   1:  PR[GP1:91,1] = PR[GP1:90,1] + -10.638;
   1:  PR[GP1:91,2] = PR[GP1:90,2] + 34.723;
   1:L PR[91] 10mm/sec CNT100;
   1:  PR[GP1:91,1] = PR[GP1:90,1] + -15.376;
   1:  PR[GP1:91,2] = PR[GP1:90,2] + 36.085;
   1:L PR[91] 10mm/sec CNT100;
   1:  PR[GP1:91,1] = PR[GP1:90,1] + -20.922;
   1:  PR[GP1:91,2] = PR[GP1:90,2] + 37.394;
   1:L PR[91] 10mm/sec CNT100;
   1:  PR[GP1:91,1] = PR[GP1:90,1] + -26.137;
   1:  PR[GP1:91,2] = PR[GP1:90,2] + 37.739;
   1:L PR[91] 10mm/sec CNT100;
   1:  PR[GP1:91,1] = PR[GP1:90,1] + -31.979;
   1:  PR[GP1:91,2] = PR[GP1:90,2] + 36.930;
   1:L PR[91] 10mm/sec CNT100;
   1:  PR[GP1:91,1] = PR[GP1:90,1] + -36.500;
   1:  PR[GP1:91,2] = PR[GP1:90,2] + 36.505;
   1:L PR[91] 10mm/sec CNT100;
   1:  PR[GP1:91,1] = PR[GP1:90,1] + -42.224;
   1:  PR[GP1:91,2] = PR[GP1:90,2] + 34.409;
   1:L PR[91] 10mm/sec CNT100;
   1:  PR[GP1:91,1] = PR[GP1:90,1] + -45.685;
   1:  PR[GP1:91,2] = PR[GP1:90,2] + 32.896;
   1:L PR[91] 10mm/sec CNT100;
   1:  PR[GP1:91,1] = PR[GP1:90,1] + -50.990;
   1:  PR[GP1:91,2] = PR[GP1:90,2] + 29.551;
   1:L PR[91] 10mm/sec CNT100;
   1:  PR[GP1:91,1] = PR[GP1:90,1] + -55.793;
   1:  PR[GP1:91,2] = PR[GP1:90,2] + 24.861;
   1:L PR[91] 10mm/sec CNT100;
   1:  PR[GP1:91,1] = PR[GP1:90,1] + -57.811;
   1:  PR[GP1:91,2] = PR[GP1:90,2] + 23.034;
   1:L PR[91] 10mm/sec CNT100;
   1:  PR[GP1:91,1] = PR[GP1:90,1] + -61.510;
   1:  PR[GP1:91,2] = PR[GP1:90,2] + 17.261;
   1:L PR[91] 10mm/sec CNT100;
   1:  PR[GP1:91,1] = PR[GP1:90,1] + -62.600;
   1:  PR[GP1:91,2] = PR[GP1:90,2] + 15.293;
   1:L PR[91] 10mm/sec CNT100;
   1:  PR[GP1:91,1] = PR[GP1:90,1] + -64.933;
   1:  PR[GP1:91,2] = PR[GP1:90,2] + 8.866;
   1:L PR[91] 10mm/sec CNT100;
   1:  PR[GP1:91,1] = PR[GP1:90,1] + -65.686;
   1:  PR[GP1:91,2] = PR[GP1:90,2] + 2.142;
   1:L PR[91] 10mm/sec CNT100;
   1:  PR[GP1:91,1] = PR[GP1:90,1] + -66.007;
   1:  PR[GP1:91,2] = PR[GP1:90,2] + 0.261;
   1:L PR[91] 10mm/sec CNT100;
   1:  PR[GP1:91,1] = PR[GP1:90,1] + -65.270;
   1:  PR[GP1:91,2] = PR[GP1:90,2] + -6.357;
   1:L PR[91] 10mm/sec CNT100;
   1:  PR[GP1:91,1] = PR[GP1:90,1] + -64.940;
   1:  PR[GP1:91,2] = PR[GP1:90,2] + -8.287;
   1:L PR[91] 10mm/sec CNT100;
   1:  PR[GP1:91,1] = PR[GP1:90,1] + -62.601;
   1:  PR[GP1:91,2] = PR[GP1:90,2] + -14.731;
   1:L PR[91] 10mm/sec CNT100;
   1:  PR[GP1:91,1] = PR[GP1:90,1] + -61.517;
   1:  PR[GP1:91,2] = PR[GP1:90,2] + -16.695;
   1:L PR[91] 10mm/sec CNT100;
   1:  PR[GP1:91,1] = PR[GP1:90,1] + -57.812;
   1:  PR[GP1:91,2] = PR[GP1:90,2] + -22.477;
   1:L PR[91] 10mm/sec CNT100;
   1:  PR[GP1:91,1] = PR[GP1:90,1] + -53.300;
   1:  PR[GP1:91,2] = PR[GP1:90,2] + -26.904;
   1:L PR[91] 10mm/sec CNT100;
   1:  PR[GP1:91,1] = PR[GP1:90,1] + -51.017;
   1:  PR[GP1:91,2] = PR[GP1:90,2] + -28.975;
   1:L PR[91] 10mm/sec CNT100;
   1:  PR[GP1:91,1] = PR[GP1:90,1] + -45.704;
   1:  PR[GP1:91,2] = PR[GP1:90,2] + -32.325;
   1:L PR[91] 10mm/sec CNT100;
   1:  PR[GP1:91,1] = PR[GP1:90,1] + -42.257;
   1:  PR[GP1:91,2] = PR[GP1:90,2] + -33.842;
   1:L PR[91] 10mm/sec CNT100;
   1:  PR[GP1:91,1] = PR[GP1:90,1] + -36.523;
   1:  PR[GP1:91,2] = PR[GP1:90,2] + -35.942;
   1:L PR[91] 10mm/sec CNT100;
   1:  PR[GP1:91,1] = PR[GP1:90,1] + -31.071;
   1:  PR[GP1:91,2] = PR[GP1:90,2] + -36.718;
   1:L PR[91] 10mm/sec CNT100;
   1:  PR[GP1:91,1] = PR[GP1:90,1] + -26.206;
   1:  PR[GP1:91,2] = PR[GP1:90,2] + -37.185;
   1:L PR[91] 10mm/sec CNT100;
   1:  PR[GP1:91,1] = PR[GP1:90,1] + -20.979;
   1:  PR[GP1:91,2] = PR[GP1:90,2] + -36.840;
   1:L PR[91] 10mm/sec CNT100;
   1:  PR[GP1:91,1] = PR[GP1:90,1] + -15.524;
   1:  PR[GP1:91,2] = PR[GP1:90,2] + -35.592;
   1:L PR[91] 10mm/sec CNT100;
   1:  PR[GP1:91,1] = PR[GP1:90,1] + -10.757;
   1:  PR[GP1:91,2] = PR[GP1:90,2] + -34.223;
   1:L PR[91] 10mm/sec CNT100;
   1:  PR[GP1:91,1] = PR[GP1:90,1] + -5.971;
   1:  PR[GP1:91,2] = PR[GP1:90,2] + -31.419;
   1:L PR[91] 10mm/sec CNT100;
   1:  PR[GP1:91,1] = PR[GP1:90,1] + -3.818;
   1:  PR[GP1:91,2] = PR[GP1:90,2] + -30.247;
   1:L PR[91] 10mm/sec CNT100;
   1:  PR[GP1:91,1] = PR[GP1:90,1] + -0.263;
   1:  PR[GP1:91,2] = PR[GP1:90,2] + -27.179;
   1:L PR[91] 10mm/sec CNT100;
   1:  PR[GP1:91,1] = PR[GP1:90,1] + 3.052;
   1:  PR[GP1:91,2] = PR[GP1:90,2] + -30.324;
   1:  PR[GP1:91,3] = PR[GP1:90,3] + 60.695;
   1:L PR[91] 10mm/sec CNT100;
   1:  PR[GP1:91,1] = PR[GP1:90,1] + 5.026;
   1:  PR[GP1:91,2] = PR[GP1:90,2] + -31.395;
   1:L PR[91] 10mm/sec CNT100;
   1:  PR[GP1:91,1] = PR[GP1:90,1] + 9.972;
   1:  PR[GP1:91,2] = PR[GP1:90,2] + -34.290;
   1:L PR[91] 10mm/sec CNT100;
   1:  PR[GP1:91,1] = PR[GP1:90,1] + 14.624;
   1:  PR[GP1:91,2] = PR[GP1:90,2] + -35.626;
   1:L PR[91] 10mm/sec CNT100;
   1:  PR[GP1:91,1] = PR[GP1:90,1] + 20.278;
   1:  PR[GP1:91,2] = PR[GP1:90,2] + -36.920;
   1:L PR[91] 10mm/sec CNT100;
   1:  PR[GP1:91,1] = PR[GP1:90,1] + 25.353;
   1:  PR[GP1:91,2] = PR[GP1:90,2] + -37.257;
   1:L PR[91] 10mm/sec CNT100;
   1:  PR[GP1:91,1] = PR[GP1:90,1] + 31.035;
   1:  PR[GP1:91,2] = PR[GP1:90,2] + -36.473;
   1:L PR[91] 10mm/sec CNT100;
   1:  PR[GP1:91,1] = PR[GP1:90,1] + 35.762;
   1:  PR[GP1:91,2] = PR[GP1:90,2] + -36.013;
   1:L PR[91] 10mm/sec CNT100;
   1:  PR[GP1:91,1] = PR[GP1:90,1] + 41.363;
   1:  PR[GP1:91,2] = PR[GP1:90,2] + -33.969;
   1:L PR[91] 10mm/sec CNT100;
   1:  PR[GP1:91,1] = PR[GP1:90,1] + 45.011;
   1:  PR[GP1:91,2] = PR[GP1:90,2] + -32.365;
   1:L PR[91] 10mm/sec CNT100;
   1:  PR[GP1:91,1] = PR[GP1:90,1] + 50.172;
   1:  PR[GP1:91,2] = PR[GP1:90,2] + -29.127;
   1:L PR[91] 10mm/sec CNT100;
   1:  PR[GP1:91,1] = PR[GP1:90,1] + 54.865;
   1:  PR[GP1:91,2] = PR[GP1:90,2] + -24.552;
   1:L PR[91] 10mm/sec CNT100;
   1:  PR[GP1:91,1] = PR[GP1:90,1] + 57.047;
   1:  PR[GP1:91,2] = PR[GP1:90,2] + -22.568;
   1:L PR[91] 10mm/sec CNT100;
   1:  PR[GP1:91,1] = PR[GP1:90,1] + 60.710;
   1:  PR[GP1:91,2] = PR[GP1:90,2] + -16.886;
   1:L PR[91] 10mm/sec CNT100;
   1:  PR[GP1:91,1] = PR[GP1:90,1] + 61.903;
   1:  PR[GP1:91,2] = PR[GP1:90,2] + -14.729;
   1:L PR[91] 10mm/sec CNT100;
   1:  PR[GP1:91,1] = PR[GP1:90,1] + 64.181;
   1:  PR[GP1:91,2] = PR[GP1:90,2] + -8.537;
   1:L PR[91] 10mm/sec CNT100;
   1:  PR[GP1:91,1] = PR[GP1:90,1] + 64.946;
   1:  PR[GP1:91,2] = PR[GP1:90,2] + -1.801;
   1:L PR[91] 10mm/sec CNT100;
   1:  PR[GP1:91,1] = PR[GP1:90,1] + 65.304;
   1:  PR[GP1:91,2] = PR[GP1:90,2] + 0.296;
   1:L PR[91] 10mm/sec CNT100;
   1:  PR[GP1:91,1] = PR[GP1:90,1] + 64.554;
   1:  PR[GP1:91,2] = PR[GP1:90,2] + 6.927;
   1:L PR[91] 10mm/sec CNT100;
   1:  PR[GP1:91,1] = PR[GP1:90,1] + 64.185;
   1:  PR[GP1:91,2] = PR[GP1:90,2] + 9.083;
   1:L PR[91] 10mm/sec CNT100;
   1:  PR[GP1:91,1] = PR[GP1:90,1] + 61.901;
   1:  PR[GP1:91,2] = PR[GP1:90,2] + 15.292;
   1:L PR[91] 10mm/sec CNT100;
   1:  PR[GP1:91,1] = PR[GP1:90,1] + 60.703;
   1:  PR[GP1:91,2] = PR[GP1:90,2] + 17.452;
   1:L PR[91] 10mm/sec CNT100;
   1:  PR[GP1:91,1] = PR[GP1:90,1] + 57.033;
   1:  PR[GP1:91,2] = PR[GP1:90,2] + 23.145;
   1:L PR[91] 10mm/sec CNT100;
   1:  PR[GP1:91,1] = PR[GP1:90,1] + 52.617;
   1:  PR[GP1:91,2] = PR[GP1:90,2] + 27.469;
   1:L PR[91] 10mm/sec CNT100;
   1:  PR[GP1:91,1] = PR[GP1:90,1] + 50.162;
   1:  PR[GP1:91,2] = PR[GP1:90,2] + 29.691;
   1:L PR[91] 10mm/sec CNT100;
   1:  PR[GP1:91,1] = PR[GP1:90,1] + 44.991;
   1:  PR[GP1:91,2] = PR[GP1:90,2] + 32.936;
   1:L PR[91] 10mm/sec CNT100;
   1:  PR[GP1:91,1] = PR[GP1:90,1] + 41.328;
   1:  PR[GP1:91,2] = PR[GP1:90,2] + 34.536;
   1:L PR[91] 10mm/sec CNT100;
   1:  PR[GP1:91,1] = PR[GP1:90,1] + 35.711;
   1:  PR[GP1:91,2] = PR[GP1:90,2] + 36.586;
   1:L PR[91] 10mm/sec CNT100;
   1:  PR[GP1:91,1] = PR[GP1:90,1] + 30.393;
   1:  PR[GP1:91,2] = PR[GP1:90,2] + 37.340;
   1:L PR[91] 10mm/sec CNT100;
   1:  PR[GP1:91,1] = PR[GP1:90,1] + 25.308;
   1:  PR[GP1:91,2] = PR[GP1:90,2] + 37.812;
   1:L PR[91] 10mm/sec CNT100;
   1:  PR[GP1:91,1] = PR[GP1:90,1] + 20.219;
   1:  PR[GP1:91,2] = PR[GP1:90,2] + 37.474;
   1:L PR[91] 10mm/sec CNT100;
   1:  PR[GP1:91,1] = PR[GP1:90,1] + 14.472;
   1:  PR[GP1:91,2] = PR[GP1:90,2] + 36.117;
   1:L PR[91] 10mm/sec CNT100;
   1:  PR[GP1:91,1] = PR[GP1:90,1] + 9.851;
   1:  PR[GP1:91,2] = PR[GP1:90,2] + 34.788;
   1:L PR[91] 10mm/sec CNT100;
   1:  PR[GP1:91,1] = PR[GP1:90,1] + 5.551;
   1:  PR[GP1:91,2] = PR[GP1:90,2] + 32.480;
   1:L PR[91] 10mm/sec CNT100;
   1:  PR[GP1:91,1] = PR[GP1:90,1] + -0.263;
   1:  PR[GP1:91,2] = PR[GP1:90,2] + 27.751;
   1:L PR[91] 10mm/sec CNT100;
   1:  PR[GP1:91,1] = PR[GP1:90,1] + -6.062;
   1:  PR[GP1:91,2] = PR[GP1:90,2] + 32.466;
   1:L PR[91] 10mm/sec CNT100;
   1:  PR[GP1:91,1] = PR[GP1:90,1] + -10.379;
   1:  PR[GP1:91,2] = PR[GP1:90,2] + 34.791;
   1:L PR[91] 10mm/sec CNT100;
   1:  PR[GP1:91,1] = PR[GP1:90,1] + -14.995;
   1:  PR[GP1:91,2] = PR[GP1:90,2] + 36.117;
   1:L PR[91] 10mm/sec CNT100;
   1:  PR[GP1:91,1] = PR[GP1:90,1] + -20.743;
   1:  PR[GP1:91,2] = PR[GP1:90,2] + 37.475;
   1:L PR[91] 10mm/sec CNT100;
   1:  PR[GP1:91,1] = PR[GP1:90,1] + -25.835;
   1:  PR[GP1:91,2] = PR[GP1:90,2] + 37.810;
   1:L PR[91] 10mm/sec CNT100;
   1:  PR[GP1:91,1] = PR[GP1:90,1] + -31.540;
   1:  PR[GP1:91,2] = PR[GP1:90,2] + 37.021;
   1:L PR[91] 10mm/sec CNT100;
   1:  PR[GP1:91,1] = PR[GP1:90,1] + -36.280;
   1:  PR[GP1:91,2] = PR[GP1:90,2] + 36.575;
   1:L PR[91] 10mm/sec CNT100;
   1:  PR[GP1:91,1] = PR[GP1:90,1] + -41.877;
   1:  PR[GP1:91,2] = PR[GP1:90,2] + 34.525;
   1:L PR[91] 10mm/sec CNT100;
   1:  PR[GP1:91,1] = PR[GP1:90,1] + -45.538;
   1:  PR[GP1:91,2] = PR[GP1:90,2] + 32.925;
   1:L PR[91] 10mm/sec CNT100;
   1:  PR[GP1:91,1] = PR[GP1:90,1] + -50.732;
   1:  PR[GP1:91,2] = PR[GP1:90,2] + 29.650;
   1:L PR[91] 10mm/sec CNT100;
   1:  PR[GP1:91,1] = PR[GP1:90,1] + -55.436;
   1:  PR[GP1:91,2] = PR[GP1:90,2] + 25.058;
   1:L PR[91] 10mm/sec CNT100;
   1:  PR[GP1:91,1] = PR[GP1:90,1] + -57.623;
   1:  PR[GP1:91,2] = PR[GP1:90,2] + 23.078;
   1:L PR[91] 10mm/sec CNT100;
   1:  PR[GP1:91,1] = PR[GP1:90,1] + -61.248;
   1:  PR[GP1:91,2] = PR[GP1:90,2] + 17.420;
   1:L PR[91] 10mm/sec CNT100;
   1:  PR[GP1:91,1] = PR[GP1:90,1] + -62.445;
   1:  PR[GP1:91,2] = PR[GP1:90,2] + 15.257;
   1:L PR[91] 10mm/sec CNT100;
   1:  PR[GP1:91,1] = PR[GP1:90,1] + -64.732;
   1:  PR[GP1:91,2] = PR[GP1:90,2] + 8.956;
   1:L PR[91] 10mm/sec CNT100;
   1:  PR[GP1:91,1] = PR[GP1:90,1] + -65.471;
   1:  PR[GP1:91,2] = PR[GP1:90,2] + 2.362;
   1:L PR[91] 10mm/sec CNT100;
   1:  PR[GP1:91,1] = PR[GP1:90,1] + -65.830;
   1:  PR[GP1:91,2] = PR[GP1:90,2] + 0.261;
   1:L PR[91] 10mm/sec CNT100;
   1:  PR[GP1:91,1] = PR[GP1:90,1] + -65.107;
   1:  PR[GP1:91,2] = PR[GP1:90,2] + -6.229;
   1:L PR[91] 10mm/sec CNT100;
   1:  PR[GP1:91,1] = PR[GP1:90,1] + -64.740;
   1:  PR[GP1:91,2] = PR[GP1:90,2] + -8.377;
   1:L PR[91] 10mm/sec CNT100;
   1:  PR[GP1:91,1] = PR[GP1:90,1] + -62.447;
   1:  PR[GP1:91,2] = PR[GP1:90,2] + -14.694;
   1:L PR[91] 10mm/sec CNT100;
   1:  PR[GP1:91,1] = PR[GP1:90,1] + -61.255;
   1:  PR[GP1:91,2] = PR[GP1:90,2] + -16.853;
   1:L PR[91] 10mm/sec CNT100;
   1:  PR[GP1:91,1] = PR[GP1:90,1] + -57.624;
   1:  PR[GP1:91,2] = PR[GP1:90,2] + -22.520;
   1:L PR[91] 10mm/sec CNT100;
   1:  PR[GP1:91,1] = PR[GP1:90,1] + -53.202;
   1:  PR[GP1:91,2] = PR[GP1:90,2] + -26.858;
   1:L PR[91] 10mm/sec CNT100;
   1:  PR[GP1:91,1] = PR[GP1:90,1] + -50.760;
   1:  PR[GP1:91,2] = PR[GP1:90,2] + -29.074;
   1:L PR[91] 10mm/sec CNT100;
   1:  PR[GP1:91,1] = PR[GP1:90,1] + -45.558;
   1:  PR[GP1:91,2] = PR[GP1:90,2] + -32.353;
   1:L PR[91] 10mm/sec CNT100;
   1:  PR[GP1:91,1] = PR[GP1:90,1] + -41.912;
   1:  PR[GP1:91,2] = PR[GP1:90,2] + -33.958;
   1:L PR[91] 10mm/sec CNT100;
   1:  PR[GP1:91,1] = PR[GP1:90,1] + -36.305;
   1:  PR[GP1:91,2] = PR[GP1:90,2] + -36.012;
   1:L PR[91] 10mm/sec CNT100;
   1:  PR[GP1:91,1] = PR[GP1:90,1] + -30.973;
   1:  PR[GP1:91,2] = PR[GP1:90,2] + -36.771;
   1:L PR[91] 10mm/sec CNT100;
   1:  PR[GP1:91,1] = PR[GP1:90,1] + -25.905;
   1:  PR[GP1:91,2] = PR[GP1:90,2] + -37.257;
   1:L PR[91] 10mm/sec CNT100;
   1:  PR[GP1:91,1] = PR[GP1:90,1] + -20.802;
   1:  PR[GP1:91,2] = PR[GP1:90,2] + -36.920;
   1:L PR[91] 10mm/sec CNT100;
   1:  PR[GP1:91,1] = PR[GP1:90,1] + -15.149;
   1:  PR[GP1:91,2] = PR[GP1:90,2] + -35.627;
   1:L PR[91] 10mm/sec CNT100;
   1:  PR[GP1:91,1] = PR[GP1:90,1] + -10.503;
   1:  PR[GP1:91,2] = PR[GP1:90,2] + -34.292;
   1:L PR[91] 10mm/sec CNT100;
   1:  PR[GP1:91,1] = PR[GP1:90,1] + -5.560;
   1:  PR[GP1:91,2] = PR[GP1:90,2] + -31.397;
   1:L PR[91] 10mm/sec CNT100;
   1:  PR[GP1:91,1] = PR[GP1:90,1] + -3.575;
   1:  PR[GP1:91,2] = PR[GP1:90,2] + -30.316;
   1:L PR[91] 10mm/sec CNT100;
   1:  PR[GP1:91,1] = PR[GP1:90,1] + -0.263;
   1:  PR[GP1:91,2] = PR[GP1:90,2] + -27.459;
   1:L PR[91] 10mm/sec CNT100;
   1:  PR[GP1:91,1] = PR[GP1:90,1] + 2.808;
   1:  PR[GP1:91,2] = PR[GP1:90,2] + -30.392;
   1:  PR[GP1:91,3] = PR[GP1:90,3] + 61.305;
   1:L PR[91] 10mm/sec CNT100;
   1:  PR[GP1:91,1] = PR[GP1:90,1] + 4.615;
   1:  PR[GP1:91,2] = PR[GP1:90,2] + -31.374;
   1:L PR[91] 10mm/sec CNT100;
   1:  PR[GP1:91,1] = PR[GP1:90,1] + 9.717;
   1:  PR[GP1:91,2] = PR[GP1:90,2] + -34.360;
   1:L PR[91] 10mm/sec CNT100;
   1:  PR[GP1:91,1] = PR[GP1:90,1] + 14.249;
   1:  PR[GP1:91,2] = PR[GP1:90,2] + -35.661;
   1:L PR[91] 10mm/sec CNT100;
   1:  PR[GP1:91,1] = PR[GP1:90,1] + 20.101;
   1:  PR[GP1:91,2] = PR[GP1:90,2] + -37.000;
   1:L PR[91] 10mm/sec CNT100;
   1:  PR[GP1:91,1] = PR[GP1:90,1] + 25.053;
   1:  PR[GP1:91,2] = PR[GP1:90,2] + -37.329;
   1:L PR[91] 10mm/sec CNT100;
   1:  PR[GP1:91,1] = PR[GP1:90,1] + 30.599;
   1:  PR[GP1:91,2] = PR[GP1:90,2] + -36.563;
   1:L PR[91] 10mm/sec CNT100;
   1:  PR[GP1:91,1] = PR[GP1:90,1] + 35.544;
   1:  PR[GP1:91,2] = PR[GP1:90,2] + -36.083;
   1:L PR[91] 10mm/sec CNT100;
   1:  PR[GP1:91,1] = PR[GP1:90,1] + 41.019;
   1:  PR[GP1:91,2] = PR[GP1:90,2] + -34.085;
   1:L PR[91] 10mm/sec CNT100;
   1:  PR[GP1:91,1] = PR[GP1:90,1] + 44.866;
   1:  PR[GP1:91,2] = PR[GP1:90,2] + -32.393;
   1:L PR[91] 10mm/sec CNT100;
   1:  PR[GP1:91,1] = PR[GP1:90,1] + 49.916;
   1:  PR[GP1:91,2] = PR[GP1:90,2] + -29.224;
   1:L PR[91] 10mm/sec CNT100;
   1:  PR[GP1:91,1] = PR[GP1:90,1] + 54.510;
   1:  PR[GP1:91,2] = PR[GP1:90,2] + -24.747;
   1:L PR[91] 10mm/sec CNT100;
   1:  PR[GP1:91,1] = PR[GP1:90,1] + 56.860;
   1:  PR[GP1:91,2] = PR[GP1:90,2] + -22.610;
   1:L PR[91] 10mm/sec CNT100;
   1:  PR[GP1:91,1] = PR[GP1:90,1] + 60.448;
   1:  PR[GP1:91,2] = PR[GP1:90,2] + -17.043;
   1:L PR[91] 10mm/sec CNT100;
   1:  PR[GP1:91,1] = PR[GP1:90,1] + 61.749;
   1:  PR[GP1:91,2] = PR[GP1:90,2] + -14.692;
   1:L PR[91] 10mm/sec CNT100;
   1:  PR[GP1:91,1] = PR[GP1:90,1] + 63.981;
   1:  PR[GP1:91,2] = PR[GP1:90,2] + -8.624;
   1:L PR[91] 10mm/sec CNT100;
   1:  PR[GP1:91,1] = PR[GP1:90,1] + 64.731;
   1:  PR[GP1:91,2] = PR[GP1:90,2] + -2.021;
   1:L PR[91] 10mm/sec CNT100;
   1:  PR[GP1:91,1] = PR[GP1:90,1] + 65.127;
   1:  PR[GP1:91,2] = PR[GP1:90,2] + 0.296;
   1:L PR[91] 10mm/sec CNT100;
   1:  PR[GP1:91,1] = PR[GP1:90,1] + 64.392;
   1:  PR[GP1:91,2] = PR[GP1:90,2] + 6.797;
   1:L PR[91] 10mm/sec CNT100;
   1:  PR[GP1:91,1] = PR[GP1:90,1] + 63.985;
   1:  PR[GP1:91,2] = PR[GP1:90,2] + 9.171;
   1:L PR[91] 10mm/sec CNT100;
   1:  PR[GP1:91,1] = PR[GP1:90,1] + 61.747;
   1:  PR[GP1:91,2] = PR[GP1:90,2] + 15.256;
   1:L PR[91] 10mm/sec CNT100;
   1:  PR[GP1:91,1] = PR[GP1:90,1] + 60.441;
   1:  PR[GP1:91,2] = PR[GP1:90,2] + 17.611;
   1:L PR[91] 10mm/sec CNT100;
   1:  PR[GP1:91,1] = PR[GP1:90,1] + 56.845;
   1:  PR[GP1:91,2] = PR[GP1:90,2] + 23.188;
   1:L PR[91] 10mm/sec CNT100;
   1:  PR[GP1:91,1] = PR[GP1:90,1] + 52.520;
   1:  PR[GP1:91,2] = PR[GP1:90,2] + 27.423;
   1:L PR[91] 10mm/sec CNT100;
   1:  PR[GP1:91,1] = PR[GP1:90,1] + 49.906;
   1:  PR[GP1:91,2] = PR[GP1:90,2] + 29.789;
   1:L PR[91] 10mm/sec CNT100;
   1:  PR[GP1:91,1] = PR[GP1:90,1] + 44.844;
   1:  PR[GP1:91,2] = PR[GP1:90,2] + 32.965;
   1:L PR[91] 10mm/sec CNT100;
   1:  PR[GP1:91,1] = PR[GP1:90,1] + 40.982;
   1:  PR[GP1:91,2] = PR[GP1:90,2] + 34.652;
   1:L PR[91] 10mm/sec CNT100;
   1:  PR[GP1:91,1] = PR[GP1:90,1] + 35.492;
   1:  PR[GP1:91,2] = PR[GP1:90,2] + 36.656;
   1:L PR[91] 10mm/sec CNT100;
   1:  PR[GP1:91,1] = PR[GP1:90,1] + 30.294;
   1:  PR[GP1:91,2] = PR[GP1:90,2] + 37.393;
   1:L PR[91] 10mm/sec CNT100;
   1:  PR[GP1:91,1] = PR[GP1:90,1] + 25.006;
   1:  PR[GP1:91,2] = PR[GP1:90,2] + 37.884;
   1:L PR[91] 10mm/sec CNT100;
   1:  PR[GP1:91,1] = PR[GP1:90,1] + 20.040;
   1:  PR[GP1:91,2] = PR[GP1:90,2] + 37.554;
   1:L PR[91] 10mm/sec CNT100;
   1:  PR[GP1:91,1] = PR[GP1:90,1] + 14.092;
   1:  PR[GP1:91,2] = PR[GP1:90,2] + 36.149;
   1:L PR[91] 10mm/sec CNT100;
   1:  PR[GP1:91,1] = PR[GP1:90,1] + 9.593;
   1:  PR[GP1:91,2] = PR[GP1:90,2] + 34.856;
   1:L PR[91] 10mm/sec CNT100;
   1:  PR[GP1:91,1] = PR[GP1:90,1] + 5.378;
   1:  PR[GP1:91,2] = PR[GP1:90,2] + 32.594;
   1:L PR[91] 10mm/sec CNT100;
   1:  PR[GP1:91,1] = PR[GP1:90,1] + -0.263;
   1:  PR[GP1:91,2] = PR[GP1:90,2] + 28.006;
   1:L PR[91] 10mm/sec CNT100;
   1:  PR[GP1:91,1] = PR[GP1:90,1] + -5.889;
   1:  PR[GP1:91,2] = PR[GP1:90,2] + 32.580;
   1:L PR[91] 10mm/sec CNT100;
   1:  PR[GP1:91,1] = PR[GP1:90,1] + -10.121;
   1:  PR[GP1:91,2] = PR[GP1:90,2] + 34.858;
   1:L PR[91] 10mm/sec CNT100;
   1:  PR[GP1:91,1] = PR[GP1:90,1] + -14.614;
   1:  PR[GP1:91,2] = PR[GP1:90,2] + 36.150;
   1:L PR[91] 10mm/sec CNT100;
   1:  PR[GP1:91,1] = PR[GP1:90,1] + -20.564;
   1:  PR[GP1:91,2] = PR[GP1:90,2] + 37.555;
   1:L PR[91] 10mm/sec CNT100;
   1:  PR[GP1:91,1] = PR[GP1:90,1] + -25.532;
   1:  PR[GP1:91,2] = PR[GP1:90,2] + 37.882;
   1:L PR[91] 10mm/sec CNT100;
   1:  PR[GP1:91,1] = PR[GP1:90,1] + -31.101;
   1:  PR[GP1:91,2] = PR[GP1:90,2] + 37.112;
   1:L PR[91] 10mm/sec CNT100;
   1:  PR[GP1:91,1] = PR[GP1:90,1] + -36.060;
   1:  PR[GP1:91,2] = PR[GP1:90,2] + 36.645;
   1:L PR[91] 10mm/sec CNT100;
   1:  PR[GP1:91,1] = PR[GP1:90,1] + -41.531;
   1:  PR[GP1:91,2] = PR[GP1:90,2] + 34.642;
   1:L PR[91] 10mm/sec CNT100;
   1:  PR[GP1:91,1] = PR[GP1:90,1] + -45.391;
   1:  PR[GP1:91,2] = PR[GP1:90,2] + 32.954;
   1:L PR[91] 10mm/sec CNT100;
   1:  PR[GP1:91,1] = PR[GP1:90,1] + -50.474;
   1:  PR[GP1:91,2] = PR[GP1:90,2] + 29.749;
   1:L PR[91] 10mm/sec CNT100;
   1:  PR[GP1:91,1] = PR[GP1:90,1] + -55.078;
   1:  PR[GP1:91,2] = PR[GP1:90,2] + 25.255;
   1:L PR[91] 10mm/sec CNT100;
   1:  PR[GP1:91,1] = PR[GP1:90,1] + -57.434;
   1:  PR[GP1:91,2] = PR[GP1:90,2] + 23.121;
   1:L PR[91] 10mm/sec CNT100;
   1:  PR[GP1:91,1] = PR[GP1:90,1] + -60.985;
   1:  PR[GP1:91,2] = PR[GP1:90,2] + 17.579;
   1:L PR[91] 10mm/sec CNT100;
   1:  PR[GP1:91,1] = PR[GP1:90,1] + -62.290;
   1:  PR[GP1:91,2] = PR[GP1:90,2] + 15.221;
   1:L PR[91] 10mm/sec CNT100;
   1:  PR[GP1:91,1] = PR[GP1:90,1] + -64.532;
   1:  PR[GP1:91,2] = PR[GP1:90,2] + 9.045;
   1:L PR[91] 10mm/sec CNT100;
   1:  PR[GP1:91,1] = PR[GP1:90,1] + -65.256;
   1:  PR[GP1:91,2] = PR[GP1:90,2] + 2.582;
   1:L PR[91] 10mm/sec CNT100;
   1:  PR[GP1:91,1] = PR[GP1:90,1] + -65.653;
   1:  PR[GP1:91,2] = PR[GP1:90,2] + 0.261;
   1:L PR[91] 10mm/sec CNT100;
   1:  PR[GP1:91,1] = PR[GP1:90,1] + -64.944;
   1:  PR[GP1:91,2] = PR[GP1:90,2] + -6.101;
   1:L PR[91] 10mm/sec CNT100;
   1:  PR[GP1:91,1] = PR[GP1:90,1] + -64.540;
   1:  PR[GP1:91,2] = PR[GP1:90,2] + -8.466;
   1:L PR[91] 10mm/sec CNT100;
   1:  PR[GP1:91,1] = PR[GP1:90,1] + -62.292;
   1:  PR[GP1:91,2] = PR[GP1:90,2] + -14.658;
   1:L PR[91] 10mm/sec CNT100;
   1:  PR[GP1:91,1] = PR[GP1:90,1] + -60.993;
   1:  PR[GP1:91,2] = PR[GP1:90,2] + -17.012;
   1:L PR[91] 10mm/sec CNT100;
   1:  PR[GP1:91,1] = PR[GP1:90,1] + -57.436;
   1:  PR[GP1:91,2] = PR[GP1:90,2] + -22.563;
   1:L PR[91] 10mm/sec CNT100;
   1:  PR[GP1:91,1] = PR[GP1:90,1] + -53.104;
   1:  PR[GP1:91,2] = PR[GP1:90,2] + -26.813;
   1:L PR[91] 10mm/sec CNT100;
   1:  PR[GP1:91,1] = PR[GP1:90,1] + -50.503;
   1:  PR[GP1:91,2] = PR[GP1:90,2] + -29.172;
   1:L PR[91] 10mm/sec CNT100;
   1:  PR[GP1:91,1] = PR[GP1:90,1] + -45.413;
   1:  PR[GP1:91,2] = PR[GP1:90,2] + -32.382;
   1:L PR[91] 10mm/sec CNT100;
   1:  PR[GP1:91,1] = PR[GP1:90,1] + -41.568;
   1:  PR[GP1:91,2] = PR[GP1:90,2] + -34.074;
   1:L PR[91] 10mm/sec CNT100;
   1:  PR[GP1:91,1] = PR[GP1:90,1] + -36.087;
   1:  PR[GP1:91,2] = PR[GP1:90,2] + -36.082;
   1:L PR[91] 10mm/sec CNT100;
   1:  PR[GP1:91,1] = PR[GP1:90,1] + -30.875;
   1:  PR[GP1:91,2] = PR[GP1:90,2] + -36.823;
   1:L PR[91] 10mm/sec CNT100;
   1:  PR[GP1:91,1] = PR[GP1:90,1] + -25.605;
   1:  PR[GP1:91,2] = PR[GP1:90,2] + -37.329;
   1:L PR[91] 10mm/sec CNT100;
   1:  PR[GP1:91,1] = PR[GP1:90,1] + -20.626;
   1:  PR[GP1:91,2] = PR[GP1:90,2] + -37.000;
   1:L PR[91] 10mm/sec CNT100;
   1:  PR[GP1:91,1] = PR[GP1:90,1] + -14.773;
   1:  PR[GP1:91,2] = PR[GP1:90,2] + -35.661;
   1:L PR[91] 10mm/sec CNT100;
   1:  PR[GP1:91,1] = PR[GP1:90,1] + -10.248;
   1:  PR[GP1:91,2] = PR[GP1:90,2] + -34.362;
   1:L PR[91] 10mm/sec CNT100;
   1:  PR[GP1:91,1] = PR[GP1:90,1] + -5.149;
   1:  PR[GP1:91,2] = PR[GP1:90,2] + -31.375;
   1:L PR[91] 10mm/sec CNT100;
   1:  PR[GP1:91,1] = PR[GP1:90,1] + -3.331;
   1:  PR[GP1:91,2] = PR[GP1:90,2] + -30.385;
   1:L PR[91] 10mm/sec CNT100;
   1:  PR[GP1:91,1] = PR[GP1:90,1] + -0.264;
   1:  PR[GP1:91,2] = PR[GP1:90,2] + -27.738;
   1:L PR[91] 10mm/sec CNT100;
   1:  PR[GP1:91,1] = PR[GP1:90,1] + 2.563;
   1:  PR[GP1:91,2] = PR[GP1:90,2] + -30.461;
   1:  PR[GP1:91,3] = PR[GP1:90,3] + 61.915;
   1:L PR[91] 10mm/sec CNT100;
   1:  PR[GP1:91,1] = PR[GP1:90,1] + 4.205;
   1:  PR[GP1:91,2] = PR[GP1:90,2] + -31.352;
   1:L PR[91] 10mm/sec CNT100;
   1:  PR[GP1:91,1] = PR[GP1:90,1] + 9.463;
   1:  PR[GP1:91,2] = PR[GP1:90,2] + -34.429;
   1:L PR[91] 10mm/sec CNT100;
   1:  PR[GP1:91,1] = PR[GP1:90,1] + 13.873;
   1:  PR[GP1:91,2] = PR[GP1:90,2] + -35.696;
   1:L PR[91] 10mm/sec CNT100;
   1:  PR[GP1:91,1] = PR[GP1:90,1] + 19.924;
   1:  PR[GP1:91,2] = PR[GP1:90,2] + -37.080;
   1:L PR[91] 10mm/sec CNT100;
   1:  PR[GP1:91,1] = PR[GP1:90,1] + 24.753;
   1:  PR[GP1:91,2] = PR[GP1:90,2] + -37.401;
   1:L PR[91] 10mm/sec CNT100;
   1:  PR[GP1:91,1] = PR[GP1:90,1] + 30.163;
   1:  PR[GP1:91,2] = PR[GP1:90,2] + -36.654;
   1:L PR[91] 10mm/sec CNT100;
   1:  PR[GP1:91,1] = PR[GP1:90,1] + 35.327;
   1:  PR[GP1:91,2] = PR[GP1:90,2] + -36.152;
   1:L PR[91] 10mm/sec CNT100;
   1:  PR[GP1:91,1] = PR[GP1:90,1] + 40.675;
   1:  PR[GP1:91,2] = PR[GP1:90,2] + -34.200;
   1:L PR[91] 10mm/sec CNT100;
   1:  PR[GP1:91,1] = PR[GP1:90,1] + 44.721;
   1:  PR[GP1:91,2] = PR[GP1:90,2] + -32.421;
   1:L PR[91] 10mm/sec CNT100;
   1:  PR[GP1:91,1] = PR[GP1:90,1] + 49.661;
   1:  PR[GP1:91,2] = PR[GP1:90,2] + -29.322;
   1:L PR[91] 10mm/sec CNT100;
   1:  PR[GP1:91,1] = PR[GP1:90,1] + 54.155;
   1:  PR[GP1:91,2] = PR[GP1:90,2] + -24.942;
   1:L PR[91] 10mm/sec CNT100;
   1:  PR[GP1:91,1] = PR[GP1:90,1] + 56.673;
   1:  PR[GP1:91,2] = PR[GP1:90,2] + -22.651;
   1:L PR[91] 10mm/sec CNT100;
   1:  PR[GP1:91,1] = PR[GP1:90,1] + 60.187;
   1:  PR[GP1:91,2] = PR[GP1:90,2] + -17.201;
   1:L PR[91] 10mm/sec CNT100;
   1:  PR[GP1:91,1] = PR[GP1:90,1] + 61.595;
   1:  PR[GP1:91,2] = PR[GP1:90,2] + -14.656;
   1:L PR[91] 10mm/sec CNT100;
   1:  PR[GP1:91,1] = PR[GP1:90,1] + 63.781;
   1:  PR[GP1:91,2] = PR[GP1:90,2] + -8.710;
   1:L PR[91] 10mm/sec CNT100;
   1:  PR[GP1:91,1] = PR[GP1:90,1] + 64.517;
   1:  PR[GP1:91,2] = PR[GP1:90,2] + -2.241;
   1:L PR[91] 10mm/sec CNT100;
   1:  PR[GP1:91,1] = PR[GP1:90,1] + 64.949;
   1:  PR[GP1:91,2] = PR[GP1:90,2] + 0.296;
   1:L PR[91] 10mm/sec CNT100;
   1:  PR[GP1:91,1] = PR[GP1:90,1] + 64.229;
   1:  PR[GP1:91,2] = PR[GP1:90,2] + 6.666;
   1:L PR[91] 10mm/sec CNT100;
   1:  PR[GP1:91,1] = PR[GP1:90,1] + 63.785;
   1:  PR[GP1:91,2] = PR[GP1:90,2] + 9.258;
   1:L PR[91] 10mm/sec CNT100;
   1:  PR[GP1:91,1] = PR[GP1:90,1] + 61.593;
   1:  PR[GP1:91,2] = PR[GP1:90,2] + 15.219;
   1:L PR[91] 10mm/sec CNT100;
   1:  PR[GP1:91,1] = PR[GP1:90,1] + 60.179;
   1:  PR[GP1:91,2] = PR[GP1:90,2] + 17.769;
   1:L PR[91] 10mm/sec CNT100;
   1:  PR[GP1:91,1] = PR[GP1:90,1] + 56.658;
   1:  PR[GP1:91,2] = PR[GP1:90,2] + 23.230;
   1:L PR[91] 10mm/sec CNT100;
   1:  PR[GP1:91,1] = PR[GP1:90,1] + 52.422;
   1:  PR[GP1:91,2] = PR[GP1:90,2] + 27.377;
   1:L PR[91] 10mm/sec CNT100;
   1:  PR[GP1:91,1] = PR[GP1:90,1] + 49.649;
   1:  PR[GP1:91,2] = PR[GP1:90,2] + 29.888;
   1:L PR[91] 10mm/sec CNT100;
   1:  PR[GP1:91,1] = PR[GP1:90,1] + 44.698;
   1:  PR[GP1:91,2] = PR[GP1:90,2] + 32.994;
   1:L PR[91] 10mm/sec CNT100;
   1:  PR[GP1:91,1] = PR[GP1:90,1] + 40.636;
   1:  PR[GP1:91,2] = PR[GP1:90,2] + 34.769;
   1:L PR[91] 10mm/sec CNT100;
   1:  PR[GP1:91,1] = PR[GP1:90,1] + 35.272;
   1:  PR[GP1:91,2] = PR[GP1:90,2] + 36.726;
   1:L PR[91] 10mm/sec CNT100;
   1:  PR[GP1:91,1] = PR[GP1:90,1] + 30.195;
   1:  PR[GP1:91,2] = PR[GP1:90,2] + 37.446;
   1:L PR[91] 10mm/sec CNT100;
   1:  PR[GP1:91,1] = PR[GP1:90,1] + 24.704;
   1:  PR[GP1:91,2] = PR[GP1:90,2] + 37.956;
   1:L PR[91] 10mm/sec CNT100;
   1:  PR[GP1:91,1] = PR[GP1:90,1] + 19.861;
   1:  PR[GP1:91,2] = PR[GP1:90,2] + 37.634;
   1:L PR[91] 10mm/sec CNT100;
   1:  PR[GP1:91,1] = PR[GP1:90,1] + 13.711;
   1:  PR[GP1:91,2] = PR[GP1:90,2] + 36.182;
   1:L PR[91] 10mm/sec CNT100;
   1:  PR[GP1:91,1] = PR[GP1:90,1] + 9.334;
   1:  PR[GP1:91,2] = PR[GP1:90,2] + 34.924;
   1:L PR[91] 10mm/sec CNT100;
   1:  PR[GP1:91,1] = PR[GP1:90,1] + 5.205;
   1:  PR[GP1:91,2] = PR[GP1:90,2] + 32.708;
   1:L PR[91] 10mm/sec CNT100;
   1:  PR[GP1:91,1] = PR[GP1:90,1] + -0.263;
   1:  PR[GP1:91,2] = PR[GP1:90,2] + 28.260;
   1:L PR[91] 10mm/sec CNT100;
   1:  PR[GP1:91,1] = PR[GP1:90,1] + -5.717;
   1:  PR[GP1:91,2] = PR[GP1:90,2] + 32.695;
   1:L PR[91] 10mm/sec CNT100;
   1:  PR[GP1:91,1] = PR[GP1:90,1] + -9.863;
   1:  PR[GP1:91,2] = PR[GP1:90,2] + 34.926;
   1:L PR[91] 10mm/sec CNT100;
   1:  PR[GP1:91,1] = PR[GP1:90,1] + -14.233;
   1:  PR[GP1:91,2] = PR[GP1:90,2] + 36.182;
   1:L PR[91] 10mm/sec CNT100;
   1:  PR[GP1:91,1] = PR[GP1:90,1] + -20.386;
   1:  PR[GP1:91,2] = PR[GP1:90,2] + 37.635;
   1:L PR[91] 10mm/sec CNT100;
   1:  PR[GP1:91,1] = PR[GP1:90,1] + -25.230;
   1:  PR[GP1:91,2] = PR[GP1:90,2] + 37.954;
   1:L PR[91] 10mm/sec CNT100;
   1:  PR[GP1:91,1] = PR[GP1:90,1] + -30.661;
   1:  PR[GP1:91,2] = PR[GP1:90,2] + 37.202;
   1:L PR[91] 10mm/sec CNT100;
   1:  PR[GP1:91,1] = PR[GP1:90,1] + -35.840;
   1:  PR[GP1:91,2] = PR[GP1:90,2] + 36.716;
   1:L PR[91] 10mm/sec CNT100;
   1:  PR[GP1:91,1] = PR[GP1:90,1] + -41.184;
   1:  PR[GP1:91,2] = PR[GP1:90,2] + 34.758;
   1:L PR[91] 10mm/sec CNT100;
   1:  PR[GP1:91,1] = PR[GP1:90,1] + -45.244;
   1:  PR[GP1:91,2] = PR[GP1:90,2] + 32.983;
   1:L PR[91] 10mm/sec CNT100;
   1:  PR[GP1:91,1] = PR[GP1:90,1] + -50.216;
   1:  PR[GP1:91,2] = PR[GP1:90,2] + 29.849;
   1:L PR[91] 10mm/sec CNT100;
   1:  PR[GP1:91,1] = PR[GP1:90,1] + -54.720;
   1:  PR[GP1:91,2] = PR[GP1:90,2] + 25.451;
   1:L PR[91] 10mm/sec CNT100;
   1:  PR[GP1:91,1] = PR[GP1:90,1] + -57.245;
   1:  PR[GP1:91,2] = PR[GP1:90,2] + 23.165;
   1:L PR[91] 10mm/sec CNT100;
   1:  PR[GP1:91,1] = PR[GP1:90,1] + -60.722;
   1:  PR[GP1:91,2] = PR[GP1:90,2] + 17.738;
   1:L PR[91] 10mm/sec CNT100;
   1:  PR[GP1:91,1] = PR[GP1:90,1] + -62.136;
   1:  PR[GP1:91,2] = PR[GP1:90,2] + 15.185;
   1:L PR[91] 10mm/sec CNT100;
   1:  PR[GP1:91,1] = PR[GP1:90,1] + -64.332;
   1:  PR[GP1:91,2] = PR[GP1:90,2] + 9.135;
   1:L PR[91] 10mm/sec CNT100;
   1:  PR[GP1:91,1] = PR[GP1:90,1] + -65.041;
   1:  PR[GP1:91,2] = PR[GP1:90,2] + 2.802;
   1:L PR[91] 10mm/sec CNT100;
   1:  PR[GP1:91,1] = PR[GP1:90,1] + -65.476;
   1:  PR[GP1:91,2] = PR[GP1:90,2] + 0.261;
   1:L PR[91] 10mm/sec CNT100;
   1:  PR[GP1:91,1] = PR[GP1:90,1] + -64.781;
   1:  PR[GP1:91,2] = PR[GP1:90,2] + -5.973;
   1:L PR[91] 10mm/sec CNT100;
   1:  PR[GP1:91,1] = PR[GP1:90,1] + -64.340;
   1:  PR[GP1:91,2] = PR[GP1:90,2] + -8.555;
   1:L PR[91] 10mm/sec CNT100;
   1:  PR[GP1:91,1] = PR[GP1:90,1] + -62.138;
   1:  PR[GP1:91,2] = PR[GP1:90,2] + -14.622;
   1:L PR[91] 10mm/sec CNT100;
   1:  PR[GP1:91,1] = PR[GP1:90,1] + -60.730;
   1:  PR[GP1:91,2] = PR[GP1:90,2] + -17.170;
   1:L PR[91] 10mm/sec CNT100;
   1:  PR[GP1:91,1] = PR[GP1:90,1] + -57.248;
   1:  PR[GP1:91,2] = PR[GP1:90,2] + -22.606;
   1:L PR[91] 10mm/sec CNT100;
   1:  PR[GP1:91,1] = PR[GP1:90,1] + -53.006;
   1:  PR[GP1:91,2] = PR[GP1:90,2] + -26.767;
   1:L PR[91] 10mm/sec CNT100;
   1:  PR[GP1:91,1] = PR[GP1:90,1] + -50.247;
   1:  PR[GP1:91,2] = PR[GP1:90,2] + -29.271;
   1:L PR[91] 10mm/sec CNT100;
   1:  PR[GP1:91,1] = PR[GP1:90,1] + -45.267;
   1:  PR[GP1:91,2] = PR[GP1:90,2] + -32.410;
   1:L PR[91] 10mm/sec CNT100;
   1:  PR[GP1:91,1] = PR[GP1:90,1] + -41.223;
   1:  PR[GP1:91,2] = PR[GP1:90,2] + -34.190;
   1:L PR[91] 10mm/sec CNT100;
   1:  PR[GP1:91,1] = PR[GP1:90,1] + -35.869;
   1:  PR[GP1:91,2] = PR[GP1:90,2] + -36.152;
   1:L PR[91] 10mm/sec CNT100;
   1:  PR[GP1:91,1] = PR[GP1:90,1] + -30.777;
   1:  PR[GP1:91,2] = PR[GP1:90,2] + -36.876;
   1:L PR[91] 10mm/sec CNT100;
   1:  PR[GP1:91,1] = PR[GP1:90,1] + -25.305;
   1:  PR[GP1:91,2] = PR[GP1:90,2] + -37.401;
   1:L PR[91] 10mm/sec CNT100;
   1:  PR[GP1:91,1] = PR[GP1:90,1] + -20.449;
   1:  PR[GP1:91,2] = PR[GP1:90,2] + -37.081;
   1:L PR[91] 10mm/sec CNT100;
   1:  PR[GP1:91,1] = PR[GP1:90,1] + -14.398;
   1:  PR[GP1:91,2] = PR[GP1:90,2] + -35.696;
   1:L PR[91] 10mm/sec CNT100;
   1:  PR[GP1:91,1] = PR[GP1:90,1] + -9.993;
   1:  PR[GP1:91,2] = PR[GP1:90,2] + -34.431;
   1:L PR[91] 10mm/sec CNT100;
   1:  PR[GP1:91,1] = PR[GP1:90,1] + -4.739;
   1:  PR[GP1:91,2] = PR[GP1:90,2] + -31.353;
   1:L PR[91] 10mm/sec CNT100;
   1:  PR[GP1:91,1] = PR[GP1:90,1] + -3.088;
   1:  PR[GP1:91,2] = PR[GP1:90,2] + -30.454;
   1:L PR[91] 10mm/sec CNT100;
   1:  PR[GP1:91,1] = PR[GP1:90,1] + -0.264;
   1:  PR[GP1:91,2] = PR[GP1:90,2] + -28.017;
   1:L PR[91] 10mm/sec CNT100;
   1:  PR[GP1:91,1] = PR[GP1:90,1] + 2.319;
   1:  PR[GP1:91,2] = PR[GP1:90,2] + -30.529;
   1:  PR[GP1:91,3] = PR[GP1:90,3] + 62.525;
   1:L PR[91] 10mm/sec CNT100;
   1:  PR[GP1:91,1] = PR[GP1:90,1] + 3.794;
   1:  PR[GP1:91,2] = PR[GP1:90,2] + -31.330;
   1:L PR[91] 10mm/sec CNT100;
   1:  PR[GP1:91,1] = PR[GP1:90,1] + 9.208;
   1:  PR[GP1:91,2] = PR[GP1:90,2] + -34.498;
   1:L PR[91] 10mm/sec CNT100;
   1:  PR[GP1:91,1] = PR[GP1:90,1] + 13.498;
   1:  PR[GP1:91,2] = PR[GP1:90,2] + -35.731;
   1:L PR[91] 10mm/sec CNT100;
   1:  PR[GP1:91,1] = PR[GP1:90,1] + 19.748;
   1:  PR[GP1:91,2] = PR[GP1:90,2] + -37.161;
   1:L PR[91] 10mm/sec CNT100;
   1:  PR[GP1:91,1] = PR[GP1:90,1] + 24.453;
   1:  PR[GP1:91,2] = PR[GP1:90,2] + -37.473;
   1:L PR[91] 10mm/sec CNT100;
   1:  PR[GP1:91,1] = PR[GP1:90,1] + 29.727;
   1:  PR[GP1:91,2] = PR[GP1:90,2] + -36.745;
   1:L PR[91] 10mm/sec CNT100;
   1:  PR[GP1:91,1] = PR[GP1:90,1] + 35.109;
   1:  PR[GP1:91,2] = PR[GP1:90,2] + -36.222;
   1:L PR[91] 10mm/sec CNT100;
   1:  PR[GP1:91,1] = PR[GP1:90,1] + 40.331;
   1:  PR[GP1:91,2] = PR[GP1:90,2] + -34.316;
   1:L PR[91] 10mm/sec CNT100;
   1:  PR[GP1:91,1] = PR[GP1:90,1] + 44.576;
   1:  PR[GP1:91,2] = PR[GP1:90,2] + -32.449;
   1:L PR[91] 10mm/sec CNT100;
   1:  PR[GP1:91,1] = PR[GP1:90,1] + 49.405;
   1:  PR[GP1:91,2] = PR[GP1:90,2] + -29.419;
   1:L PR[91] 10mm/sec CNT100;
   1:  PR[GP1:91,1] = PR[GP1:90,1] + 53.800;
   1:  PR[GP1:91,2] = PR[GP1:90,2] + -25.136;
   1:L PR[91] 10mm/sec CNT100;
   1:  PR[GP1:91,1] = PR[GP1:90,1] + 56.486;
   1:  PR[GP1:91,2] = PR[GP1:90,2] + -22.693;
   1:L PR[91] 10mm/sec CNT100;
   1:  PR[GP1:91,1] = PR[GP1:90,1] + 59.925;
   1:  PR[GP1:91,2] = PR[GP1:90,2] + -17.358;
   1:L PR[91] 10mm/sec CNT100;
   1:  PR[GP1:91,1] = PR[GP1:90,1] + 61.441;
   1:  PR[GP1:91,2] = PR[GP1:90,2] + -14.619;
   1:L PR[91] 10mm/sec CNT100;
   1:  PR[GP1:91,1] = PR[GP1:90,1] + 63.582;
   1:  PR[GP1:91,2] = PR[GP1:90,2] + -8.797;
   1:L PR[91] 10mm/sec CNT100;
   1:  PR[GP1:91,1] = PR[GP1:90,1] + 64.302;
   1:  PR[GP1:91,2] = PR[GP1:90,2] + -2.461;
   1:L PR[91] 10mm/sec CNT100;
   1:  PR[GP1:91,1] = PR[GP1:90,1] + 64.772;
   1:  PR[GP1:91,2] = PR[GP1:90,2] + 0.296;
   1:L PR[91] 10mm/sec CNT100;
   1:  PR[GP1:91,1] = PR[GP1:90,1] + 64.067;
   1:  PR[GP1:91,2] = PR[GP1:90,2] + 6.535;
   1:L PR[91] 10mm/sec CNT100;
   1:  PR[GP1:91,1] = PR[GP1:90,1] + 63.586;
   1:  PR[GP1:91,2] = PR[GP1:90,2] + 9.345;
   1:L PR[91] 10mm/sec CNT100;
   1:  PR[GP1:91,1] = PR[GP1:90,1] + 61.439;
   1:  PR[GP1:91,2] = PR[GP1:90,2] + 15.183;
   1:L PR[91] 10mm/sec CNT100;
   1:  PR[GP1:91,1] = PR[GP1:90,1] + 59.916;
   1:  PR[GP1:91,2] = PR[GP1:90,2] + 17.927;
   1:L PR[91] 10mm/sec CNT100;
   1:  PR[GP1:91,1] = PR[GP1:90,1] + 56.470;
   1:  PR[GP1:91,2] = PR[GP1:90,2] + 23.272;
   1:L PR[91] 10mm/sec CNT100;
   1:  PR[GP1:91,1] = PR[GP1:90,1] + 52.325;
   1:  PR[GP1:91,2] = PR[GP1:90,2] + 27.331;
   1:L PR[91] 10mm/sec CNT100;
   1:  PR[GP1:91,1] = PR[GP1:90,1] + 49.392;
   1:  PR[GP1:91,2] = PR[GP1:90,2] + 29.986;
   1:L PR[91] 10mm/sec CNT100;
   1:  PR[GP1:91,1] = PR[GP1:90,1] + 44.552;
   1:  PR[GP1:91,2] = PR[GP1:90,2] + 33.023;
   1:L PR[91] 10mm/sec CNT100;
   1:  PR[GP1:91,1] = PR[GP1:90,1] + 40.290;
   1:  PR[GP1:91,2] = PR[GP1:90,2] + 34.885;
   1:L PR[91] 10mm/sec CNT100;
   1:  PR[GP1:91,1] = PR[GP1:90,1] + 35.053;
   1:  PR[GP1:91,2] = PR[GP1:90,2] + 36.796;
   1:L PR[91] 10mm/sec CNT100;
   1:  PR[GP1:91,1] = PR[GP1:90,1] + 30.096;
   1:  PR[GP1:91,2] = PR[GP1:90,2] + 37.499;
   1:L PR[91] 10mm/sec CNT100;
   1:  PR[GP1:91,1] = PR[GP1:90,1] + 24.402;
   1:  PR[GP1:91,2] = PR[GP1:90,2] + 38.028;
   1:L PR[91] 10mm/sec CNT100;
   1:  PR[GP1:91,1] = PR[GP1:90,1] + 19.683;
   1:  PR[GP1:91,2] = PR[GP1:90,2] + 37.714;
   1:L PR[91] 10mm/sec CNT100;
   1:  PR[GP1:91,1] = PR[GP1:90,1] + 13.330;
   1:  PR[GP1:91,2] = PR[GP1:90,2] + 36.214;
   1:L PR[91] 10mm/sec CNT100;
   1:  PR[GP1:91,1] = PR[GP1:90,1] + 9.076;
   1:  PR[GP1:91,2] = PR[GP1:90,2] + 34.991;
   1:L PR[91] 10mm/sec CNT100;
   1:  PR[GP1:91,1] = PR[GP1:90,1] + 5.032;
   1:  PR[GP1:91,2] = PR[GP1:90,2] + 32.822;
   1:L PR[91] 10mm/sec CNT100;
   1:  PR[GP1:91,1] = PR[GP1:90,1] + -0.263;
   1:  PR[GP1:91,2] = PR[GP1:90,2] + 28.515;
   1:L PR[91] 10mm/sec CNT100;
   1:  PR[GP1:91,1] = PR[GP1:90,1] + -5.545;
   1:  PR[GP1:91,2] = PR[GP1:90,2] + 32.810;
   1:L PR[91] 10mm/sec CNT100;
   1:  PR[GP1:91,1] = PR[GP1:90,1] + -8.723;
   1:  PR[GP1:91,2] = PR[GP1:90,2] + 34.531;
   1:L PR[91] 10mm/sec CNT100;
   1:  PR[GP1:91,1] = PR[GP1:90,1] + -9.602;
   1:  PR[GP1:91,2] = PR[GP1:90,2] + 34.992;
   1:L PR[91] 10mm/sec CNT100;
   1:  PR[GP1:91,1] = PR[GP1:90,1] + -13.852;
   1:  PR[GP1:91,2] = PR[GP1:90,2] + 36.215;
   1:L PR[91] 10mm/sec CNT100;
   1:  PR[GP1:91,1] = PR[GP1:90,1] + -20.207;
   1:  PR[GP1:91,2] = PR[GP1:90,2] + 37.715;
   1:L PR[91] 10mm/sec CNT100;
   1:  PR[GP1:91,1] = PR[GP1:90,1] + -24.927;
   1:  PR[GP1:91,2] = PR[GP1:90,2] + 38.026;
   1:L PR[91] 10mm/sec CNT100;
   1:  PR[GP1:91,1] = PR[GP1:90,1] + -30.222;
   1:  PR[GP1:91,2] = PR[GP1:90,2] + 37.293;
   1:L PR[91] 10mm/sec CNT100;
   1:  PR[GP1:91,1] = PR[GP1:90,1] + -35.620;
   1:  PR[GP1:91,2] = PR[GP1:90,2] + 36.786;
   1:L PR[91] 10mm/sec CNT100;
   1:  PR[GP1:91,1] = PR[GP1:90,1] + -40.838;
   1:  PR[GP1:91,2] = PR[GP1:90,2] + 34.875;
   1:L PR[91] 10mm/sec CNT100;
   1:  PR[GP1:91,1] = PR[GP1:90,1] + -45.098;
   1:  PR[GP1:91,2] = PR[GP1:90,2] + 33.012;
   1:L PR[91] 10mm/sec CNT100;
   1:  PR[GP1:91,1] = PR[GP1:90,1] + -49.958;
   1:  PR[GP1:91,2] = PR[GP1:90,2] + 29.948;
   1:L PR[91] 10mm/sec CNT100;
   1:  PR[GP1:91,1] = PR[GP1:90,1] + -54.363;
   1:  PR[GP1:91,2] = PR[GP1:90,2] + 25.648;
   1:L PR[91] 10mm/sec CNT100;
   1:  PR[GP1:91,1] = PR[GP1:90,1] + -57.057;
   1:  PR[GP1:91,2] = PR[GP1:90,2] + 23.209;
   1:L PR[91] 10mm/sec CNT100;
   1:  PR[GP1:91,1] = PR[GP1:90,1] + -60.460;
   1:  PR[GP1:91,2] = PR[GP1:90,2] + 17.898;
   1:L PR[91] 10mm/sec CNT100;
   1:  PR[GP1:91,1] = PR[GP1:90,1] + -61.981;
   1:  PR[GP1:91,2] = PR[GP1:90,2] + 15.149;
   1:L PR[91] 10mm/sec CNT100;
   1:  PR[GP1:91,1] = PR[GP1:90,1] + -64.131;
   1:  PR[GP1:91,2] = PR[GP1:90,2] + 9.225;
   1:L PR[91] 10mm/sec CNT100;
   1:  PR[GP1:91,1] = PR[GP1:90,1] + -64.826;
   1:  PR[GP1:91,2] = PR[GP1:90,2] + 3.022;
   1:L PR[91] 10mm/sec CNT100;
   1:  PR[GP1:91,1] = PR[GP1:90,1] + -65.299;
   1:  PR[GP1:91,2] = PR[GP1:90,2] + 0.261;
   1:L PR[91] 10mm/sec CNT100;
   1:  PR[GP1:91,1] = PR[GP1:90,1] + -64.618;
   1:  PR[GP1:91,2] = PR[GP1:90,2] + -5.845;
   1:L PR[91] 10mm/sec CNT100;
   1:  PR[GP1:91,1] = PR[GP1:90,1] + -64.139;
   1:  PR[GP1:91,2] = PR[GP1:90,2] + -8.644;
   1:L PR[91] 10mm/sec CNT100;
   1:  PR[GP1:91,1] = PR[GP1:90,1] + -61.983;
   1:  PR[GP1:91,2] = PR[GP1:90,2] + -14.585;
   1:L PR[91] 10mm/sec CNT100;
   1:  PR[GP1:91,1] = PR[GP1:90,1] + -60.468;
   1:  PR[GP1:91,2] = PR[GP1:90,2] + -17.328;
   1:L PR[91] 10mm/sec CNT100;
   1:  PR[GP1:91,1] = PR[GP1:90,1] + -57.060;
   1:  PR[GP1:91,2] = PR[GP1:90,2] + -22.649;
   1:L PR[91] 10mm/sec CNT100;
   1:  PR[GP1:91,1] = PR[GP1:90,1] + -52.909;
   1:  PR[GP1:91,2] = PR[GP1:90,2] + -26.721;
   1:L PR[91] 10mm/sec CNT100;
   1:  PR[GP1:91,1] = PR[GP1:90,1] + -49.990;
   1:  PR[GP1:91,2] = PR[GP1:90,2] + -29.369;
   1:L PR[91] 10mm/sec CNT100;
   1:  PR[GP1:91,1] = PR[GP1:90,1] + -45.122;
   1:  PR[GP1:91,2] = PR[GP1:90,2] + -32.439;
   1:L PR[91] 10mm/sec CNT100;
   1:  PR[GP1:91,1] = PR[GP1:90,1] + -40.878;
   1:  PR[GP1:91,2] = PR[GP1:90,2] + -34.306;
   1:L PR[91] 10mm/sec CNT100;
   1:  PR[GP1:91,1] = PR[GP1:90,1] + -35.651;
   1:  PR[GP1:91,2] = PR[GP1:90,2] + -36.221;
   1:L PR[91] 10mm/sec CNT100;
   1:  PR[GP1:91,1] = PR[GP1:90,1] + -30.679;
   1:  PR[GP1:91,2] = PR[GP1:90,2] + -36.929;
   1:L PR[91] 10mm/sec CNT100;
   1:  PR[GP1:91,1] = PR[GP1:90,1] + -25.005;
   1:  PR[GP1:91,2] = PR[GP1:90,2] + -37.473;
   1:L PR[91] 10mm/sec CNT100;
   1:  PR[GP1:91,1] = PR[GP1:90,1] + -20.272;
   1:  PR[GP1:91,2] = PR[GP1:90,2] + -37.161;
   1:L PR[91] 10mm/sec CNT100;
   1:  PR[GP1:91,1] = PR[GP1:90,1] + -14.023;
   1:  PR[GP1:91,2] = PR[GP1:90,2] + -35.731;
   1:L PR[91] 10mm/sec CNT100;
   1:  PR[GP1:91,1] = PR[GP1:90,1] + -9.738;
   1:  PR[GP1:91,2] = PR[GP1:90,2] + -34.501;
   1:L PR[91] 10mm/sec CNT100;
   1:  PR[GP1:91,1] = PR[GP1:90,1] + -4.328;
   1:  PR[GP1:91,2] = PR[GP1:90,2] + -31.331;
   1:L PR[91] 10mm/sec CNT100;
   1:  PR[GP1:91,1] = PR[GP1:90,1] + -2.844;
   1:  PR[GP1:91,2] = PR[GP1:90,2] + -30.523;
   1:L PR[91] 10mm/sec CNT100;
   1:  PR[GP1:91,1] = PR[GP1:90,1] + -0.264;
   1:  PR[GP1:91,2] = PR[GP1:90,2] + -28.297;
   1:L PR[91] 10mm/sec CNT100;
   1:  PR[GP1:91,1] = PR[GP1:90,1] + 2.074;
   1:  PR[GP1:91,2] = PR[GP1:90,2] + -30.597;
   1:  PR[GP1:91,3] = PR[GP1:90,3] + 63.135;
   1:L PR[91] 10mm/sec CNT100;
   1:  PR[GP1:91,1] = PR[GP1:90,1] + 3.384;
   1:  PR[GP1:91,2] = PR[GP1:90,2] + -31.308;
   1:L PR[91] 10mm/sec CNT100;
   1:  PR[GP1:91,1] = PR[GP1:90,1] + 8.953;
   1:  PR[GP1:91,2] = PR[GP1:90,2] + -34.568;
   1:L PR[91] 10mm/sec CNT100;
   1:  PR[GP1:91,1] = PR[GP1:90,1] + 13.123;
   1:  PR[GP1:91,2] = PR[GP1:90,2] + -35.765;
   1:L PR[91] 10mm/sec CNT100;
   1:  PR[GP1:91,1] = PR[GP1:90,1] + 19.571;
   1:  PR[GP1:91,2] = PR[GP1:90,2] + -37.241;
   1:L PR[91] 10mm/sec CNT100;
   1:  PR[GP1:91,1] = PR[GP1:90,1] + 24.153;
   1:  PR[GP1:91,2] = PR[GP1:90,2] + -37.545;
   1:L PR[91] 10mm/sec CNT100;
   1:  PR[GP1:91,1] = PR[GP1:90,1] + 29.291;
   1:  PR[GP1:91,2] = PR[GP1:90,2] + -36.836;
   1:L PR[91] 10mm/sec CNT100;
   1:  PR[GP1:91,1] = PR[GP1:90,1] + 34.892;
   1:  PR[GP1:91,2] = PR[GP1:90,2] + -36.292;
   1:L PR[91] 10mm/sec CNT100;
   1:  PR[GP1:91,1] = PR[GP1:90,1] + 39.987;
   1:  PR[GP1:91,2] = PR[GP1:90,2] + -34.432;
   1:L PR[91] 10mm/sec CNT100;
   1:  PR[GP1:91,1] = PR[GP1:90,1] + 44.430;
   1:  PR[GP1:91,2] = PR[GP1:90,2] + -32.478;
   1:L PR[91] 10mm/sec CNT100;
   1:  PR[GP1:91,1] = PR[GP1:90,1] + 49.150;
   1:  PR[GP1:91,2] = PR[GP1:90,2] + -29.517;
   1:L PR[91] 10mm/sec CNT100;
   1:  PR[GP1:91,1] = PR[GP1:90,1] + 53.445;
   1:  PR[GP1:91,2] = PR[GP1:90,2] + -25.331;
   1:L PR[91] 10mm/sec CNT100;
   1:  PR[GP1:91,1] = PR[GP1:90,1] + 56.299;
   1:  PR[GP1:91,2] = PR[GP1:90,2] + -22.734;
   1:L PR[91] 10mm/sec CNT100;
   1:  PR[GP1:91,1] = PR[GP1:90,1] + 59.663;
   1:  PR[GP1:91,2] = PR[GP1:90,2] + -17.516;
   1:L PR[91] 10mm/sec CNT100;
   1:  PR[GP1:91,1] = PR[GP1:90,1] + 61.287;
   1:  PR[GP1:91,2] = PR[GP1:90,2] + -14.582;
   1:L PR[91] 10mm/sec CNT100;
   1:  PR[GP1:91,1] = PR[GP1:90,1] + 63.382;
   1:  PR[GP1:91,2] = PR[GP1:90,2] + -8.884;
   1:L PR[91] 10mm/sec CNT100;
   1:  PR[GP1:91,1] = PR[GP1:90,1] + 64.087;
   1:  PR[GP1:91,2] = PR[GP1:90,2] + -2.680;
   1:L PR[91] 10mm/sec CNT100;
   1:  PR[GP1:91,1] = PR[GP1:90,1] + 64.595;
   1:  PR[GP1:91,2] = PR[GP1:90,2] + 0.296;
   1:L PR[91] 10mm/sec CNT100;
   1:  PR[GP1:91,1] = PR[GP1:90,1] + 63.904;
   1:  PR[GP1:91,2] = PR[GP1:90,2] + 6.405;
   1:L PR[91] 10mm/sec CNT100;
   1:  PR[GP1:91,1] = PR[GP1:90,1] + 63.386;
   1:  PR[GP1:91,2] = PR[GP1:90,2] + 9.432;
   1:L PR[91] 10mm/sec CNT100;
   1:  PR[GP1:91,1] = PR[GP1:90,1] + 61.284;
   1:  PR[GP1:91,2] = PR[GP1:90,2] + 15.146;
   1:L PR[91] 10mm/sec CNT100;
   1:  PR[GP1:91,1] = PR[GP1:90,1] + 59.654;
   1:  PR[GP1:91,2] = PR[GP1:90,2] + 18.086;
   1:L PR[91] 10mm/sec CNT100;
   1:  PR[GP1:91,1] = PR[GP1:90,1] + 56.283;
   1:  PR[GP1:91,2] = PR[GP1:90,2] + 23.314;
   1:L PR[91] 10mm/sec CNT100;
   1:  PR[GP1:91,1] = PR[GP1:90,1] + 52.228;
   1:  PR[GP1:91,2] = PR[GP1:90,2] + 27.286;
   1:L PR[91] 10mm/sec CNT100;
   1:  PR[GP1:91,1] = PR[GP1:90,1] + 49.135;
   1:  PR[GP1:91,2] = PR[GP1:90,2] + 30.084;
   1:L PR[91] 10mm/sec CNT100;
   1:  PR[GP1:91,1] = PR[GP1:90,1] + 44.405;
   1:  PR[GP1:91,2] = PR[GP1:90,2] + 33.052;
   1:L PR[91] 10mm/sec CNT100;
   1:  PR[GP1:91,1] = PR[GP1:90,1] + 39.944;
   1:  PR[GP1:91,2] = PR[GP1:90,2] + 35.001;
   1:L PR[91] 10mm/sec CNT100;
   1:  PR[GP1:91,1] = PR[GP1:90,1] + 34.834;
   1:  PR[GP1:91,2] = PR[GP1:90,2] + 36.866;
   1:L PR[91] 10mm/sec CNT100;
   1:  PR[GP1:91,1] = PR[GP1:90,1] + 29.996;
   1:  PR[GP1:91,2] = PR[GP1:90,2] + 37.552;
   1:L PR[91] 10mm/sec CNT100;
   1:  PR[GP1:91,1] = PR[GP1:90,1] + 24.099;
   1:  PR[GP1:91,2] = PR[GP1:90,2] + 38.100;
   1:L PR[91] 10mm/sec CNT100;
   1:  PR[GP1:91,1] = PR[GP1:90,1] + 19.504;
   1:  PR[GP1:91,2] = PR[GP1:90,2] + 37.795;
   1:L PR[91] 10mm/sec CNT100;
   1:  PR[GP1:91,1] = PR[GP1:90,1] + 12.949;
   1:  PR[GP1:91,2] = PR[GP1:90,2] + 36.247;
   1:L PR[91] 10mm/sec CNT100;
   1:  PR[GP1:91,1] = PR[GP1:90,1] + 8.816;
   1:  PR[GP1:91,2] = PR[GP1:90,2] + 35.058;
   1:L PR[91] 10mm/sec CNT100;
   1:  PR[GP1:91,1] = PR[GP1:90,1] + 7.908;
   1:  PR[GP1:91,2] = PR[GP1:90,2] + 34.582;
   1:L PR[91] 10mm/sec CNT100;
   1:  PR[GP1:91,1] = PR[GP1:90,1] + 4.860;
   1:  PR[GP1:91,2] = PR[GP1:90,2] + 32.936;
   1:L PR[91] 10mm/sec CNT100;
   1:  PR[GP1:91,1] = PR[GP1:90,1] + -0.263;
   1:  PR[GP1:91,2] = PR[GP1:90,2] + 28.770;
   1:L PR[91] 10mm/sec CNT100;
   1:  PR[GP1:91,1] = PR[GP1:90,1] + -5.373;
   1:  PR[GP1:91,2] = PR[GP1:90,2] + 32.924;
   1:L PR[91] 10mm/sec CNT100;
   1:  PR[GP1:91,1] = PR[GP1:90,1] + -8.438;
   1:  PR[GP1:91,2] = PR[GP1:90,2] + 34.584;
   1:L PR[91] 10mm/sec CNT100;
   1:  PR[GP1:91,1] = PR[GP1:90,1] + -9.344;
   1:  PR[GP1:91,2] = PR[GP1:90,2] + 35.060;
   1:L PR[91] 10mm/sec CNT100;
   1:  PR[GP1:91,1] = PR[GP1:90,1] + -13.472;
   1:  PR[GP1:91,2] = PR[GP1:90,2] + 36.247;
   1:L PR[91] 10mm/sec CNT100;
   1:  PR[GP1:91,1] = PR[GP1:90,1] + -20.028;
   1:  PR[GP1:91,2] = PR[GP1:90,2] + 37.795;
   1:L PR[91] 10mm/sec CNT100;
   1:  PR[GP1:91,1] = PR[GP1:90,1] + -24.624;
   1:  PR[GP1:91,2] = PR[GP1:90,2] + 38.098;
   1:L PR[91] 10mm/sec CNT100;
   1:  PR[GP1:91,1] = PR[GP1:90,1] + -29.783;
   1:  PR[GP1:91,2] = PR[GP1:90,2] + 37.384;
   1:L PR[91] 10mm/sec CNT100;
   1:  PR[GP1:91,1] = PR[GP1:90,1] + -35.400;
   1:  PR[GP1:91,2] = PR[GP1:90,2] + 36.856;
   1:L PR[91] 10mm/sec CNT100;
   1:  PR[GP1:91,1] = PR[GP1:90,1] + -40.491;
   1:  PR[GP1:91,2] = PR[GP1:90,2] + 34.992;
   1:L PR[91] 10mm/sec CNT100;
   1:  PR[GP1:91,1] = PR[GP1:90,1] + -44.951;
   1:  PR[GP1:91,2] = PR[GP1:90,2] + 33.042;
   1:L PR[91] 10mm/sec CNT100;
   1:  PR[GP1:91,1] = PR[GP1:90,1] + -49.700;
   1:  PR[GP1:91,2] = PR[GP1:90,2] + 30.047;
   1:L PR[91] 10mm/sec CNT100;
   1:  PR[GP1:91,1] = PR[GP1:90,1] + -54.005;
   1:  PR[GP1:91,2] = PR[GP1:90,2] + 25.844;
   1:L PR[91] 10mm/sec CNT100;
   1:  PR[GP1:91,1] = PR[GP1:90,1] + -56.868;
   1:  PR[GP1:91,2] = PR[GP1:90,2] + 23.252;
   1:L PR[91] 10mm/sec CNT100;
   1:  PR[GP1:91,1] = PR[GP1:90,1] + -60.197;
   1:  PR[GP1:91,2] = PR[GP1:90,2] + 18.057;
   1:L PR[91] 10mm/sec CNT100;
   1:  PR[GP1:91,1] = PR[GP1:90,1] + -61.826;
   1:  PR[GP1:91,2] = PR[GP1:90,2] + 15.113;
   1:L PR[91] 10mm/sec CNT100;
   1:  PR[GP1:91,1] = PR[GP1:90,1] + -63.931;
   1:  PR[GP1:91,2] = PR[GP1:90,2] + 9.315;
   1:L PR[91] 10mm/sec CNT100;
   1:  PR[GP1:91,1] = PR[GP1:90,1] + -64.611;
   1:  PR[GP1:91,2] = PR[GP1:90,2] + 3.242;
   1:L PR[91] 10mm/sec CNT100;
   1:  PR[GP1:91,1] = PR[GP1:90,1] + -65.121;
   1:  PR[GP1:91,2] = PR[GP1:90,2] + 0.261;
   1:L PR[91] 10mm/sec CNT100;
   1:  PR[GP1:91,1] = PR[GP1:90,1] + -64.455;
   1:  PR[GP1:91,2] = PR[GP1:90,2] + -5.717;
   1:L PR[91] 10mm/sec CNT100;
   1:  PR[GP1:91,1] = PR[GP1:90,1] + -63.939;
   1:  PR[GP1:91,2] = PR[GP1:90,2] + -8.734;
   1:L PR[91] 10mm/sec CNT100;
   1:  PR[GP1:91,1] = PR[GP1:90,1] + -61.829;
   1:  PR[GP1:91,2] = PR[GP1:90,2] + -14.549;
   1:L PR[91] 10mm/sec CNT100;
   1:  PR[GP1:91,1] = PR[GP1:90,1] + -60.206;
   1:  PR[GP1:91,2] = PR[GP1:90,2] + -17.487;
   1:L PR[91] 10mm/sec CNT100;
   1:  PR[GP1:91,1] = PR[GP1:90,1] + -56.872;
   1:  PR[GP1:91,2] = PR[GP1:90,2] + -22.692;
   1:L PR[91] 10mm/sec CNT100;
   1:  PR[GP1:91,1] = PR[GP1:90,1] + -52.811;
   1:  PR[GP1:91,2] = PR[GP1:90,2] + -26.676;
   1:L PR[91] 10mm/sec CNT100;
   1:  PR[GP1:91,1] = PR[GP1:90,1] + -49.733;
   1:  PR[GP1:91,2] = PR[GP1:90,2] + -29.468;
   1:L PR[91] 10mm/sec CNT100;
   1:  PR[GP1:91,1] = PR[GP1:90,1] + -44.976;
   1:  PR[GP1:91,2] = PR[GP1:90,2] + -32.467;
   1:L PR[91] 10mm/sec CNT100;
   1:  PR[GP1:91,1] = PR[GP1:90,1] + -40.534;
   1:  PR[GP1:91,2] = PR[GP1:90,2] + -34.422;
   1:L PR[91] 10mm/sec CNT100;
   1:  PR[GP1:91,1] = PR[GP1:90,1] + -35.432;
   1:  PR[GP1:91,2] = PR[GP1:90,2] + -36.291;
   1:L PR[91] 10mm/sec CNT100;
   1:  PR[GP1:91,1] = PR[GP1:90,1] + -30.581;
   1:  PR[GP1:91,2] = PR[GP1:90,2] + -36.981;
   1:L PR[91] 10mm/sec CNT100;
   1:  PR[GP1:91,1] = PR[GP1:90,1] + -24.704;
   1:  PR[GP1:91,2] = PR[GP1:90,2] + -37.545;
   1:L PR[91] 10mm/sec CNT100;
   1:  PR[GP1:91,1] = PR[GP1:90,1] + -20.095;
   1:  PR[GP1:91,2] = PR[GP1:90,2] + -37.241;
   1:L PR[91] 10mm/sec CNT100;
   1:  PR[GP1:91,1] = PR[GP1:90,1] + -13.647;
   1:  PR[GP1:91,2] = PR[GP1:90,2] + -35.766;
   1:L PR[91] 10mm/sec CNT100;
   1:  PR[GP1:91,1] = PR[GP1:90,1] + -9.484;
   1:  PR[GP1:91,2] = PR[GP1:90,2] + -34.570;
   1:L PR[91] 10mm/sec CNT100;
   1:  PR[GP1:91,1] = PR[GP1:90,1] + -3.918;
   1:  PR[GP1:91,2] = PR[GP1:90,2] + -31.309;
   1:L PR[91] 10mm/sec CNT100;
   1:  PR[GP1:91,1] = PR[GP1:90,1] + -2.601;
   1:  PR[GP1:91,2] = PR[GP1:90,2] + -30.592;
   1:L PR[91] 10mm/sec CNT100;
   1:  PR[GP1:91,1] = PR[GP1:90,1] + -0.264;
   1:  PR[GP1:91,2] = PR[GP1:90,2] + -28.576;
   1:L PR[91] 10mm/sec CNT100;
   1:  PR[GP1:91,1] = PR[GP1:90,1] + 1.830;
   1:  PR[GP1:91,2] = PR[GP1:90,2] + -30.666;
   1:  PR[GP1:91,3] = PR[GP1:90,3] + 63.745;
   1:L PR[91] 10mm/sec CNT100;
   1:  PR[GP1:91,1] = PR[GP1:90,1] + 2.973;
   1:  PR[GP1:91,2] = PR[GP1:90,2] + -31.286;
   1:L PR[91] 10mm/sec CNT100;
   1:  PR[GP1:91,1] = PR[GP1:90,1] + 8.699;
   1:  PR[GP1:91,2] = PR[GP1:90,2] + -34.637;
   1:L PR[91] 10mm/sec CNT100;
   1:  PR[GP1:91,1] = PR[GP1:90,1] + 12.747;
   1:  PR[GP1:91,2] = PR[GP1:90,2] + -35.800;
   1:L PR[91] 10mm/sec CNT100;
   1:  PR[GP1:91,1] = PR[GP1:90,1] + 19.394;
   1:  PR[GP1:91,2] = PR[GP1:90,2] + -37.321;
   1:L PR[91] 10mm/sec CNT100;
   1:  PR[GP1:91,1] = PR[GP1:90,1] + 23.853;
   1:  PR[GP1:91,2] = PR[GP1:90,2] + -37.617;
   1:L PR[91] 10mm/sec CNT100;
   1:  PR[GP1:91,1] = PR[GP1:90,1] + 28.855;
   1:  PR[GP1:91,2] = PR[GP1:90,2] + -36.927;
   1:L PR[91] 10mm/sec CNT100;
   1:  PR[GP1:91,1] = PR[GP1:90,1] + 34.674;
   1:  PR[GP1:91,2] = PR[GP1:90,2] + -36.361;
   1:L PR[91] 10mm/sec CNT100;
   1:  PR[GP1:91,1] = PR[GP1:90,1] + 39.642;
   1:  PR[GP1:91,2] = PR[GP1:90,2] + -34.548;
   1:L PR[91] 10mm/sec CNT100;
   1:  PR[GP1:91,1] = PR[GP1:90,1] + 44.285;
   1:  PR[GP1:91,2] = PR[GP1:90,2] + -32.506;
   1:L PR[91] 10mm/sec CNT100;
   1:  PR[GP1:91,1] = PR[GP1:90,1] + 48.894;
   1:  PR[GP1:91,2] = PR[GP1:90,2] + -29.614;
   1:L PR[91] 10mm/sec CNT100;
   1:  PR[GP1:91,1] = PR[GP1:90,1] + 53.090;
   1:  PR[GP1:91,2] = PR[GP1:90,2] + -25.525;
   1:L PR[91] 10mm/sec CNT100;
   1:  PR[GP1:91,1] = PR[GP1:90,1] + 56.112;
   1:  PR[GP1:91,2] = PR[GP1:90,2] + -22.776;
   1:L PR[91] 10mm/sec CNT100;
   1:  PR[GP1:91,1] = PR[GP1:90,1] + 59.402;
   1:  PR[GP1:91,2] = PR[GP1:90,2] + -17.674;
   1:L PR[91] 10mm/sec CNT100;
   1:  PR[GP1:91,1] = PR[GP1:90,1] + 61.132;
   1:  PR[GP1:91,2] = PR[GP1:90,2] + -14.545;
   1:L PR[91] 10mm/sec CNT100;
   1:  PR[GP1:91,1] = PR[GP1:90,1] + 63.183;
   1:  PR[GP1:91,2] = PR[GP1:90,2] + -8.971;
   1:L PR[91] 10mm/sec CNT100;
   1:  PR[GP1:91,1] = PR[GP1:90,1] + 63.873;
   1:  PR[GP1:91,2] = PR[GP1:90,2] + -2.900;
   1:L PR[91] 10mm/sec CNT100;
   1:  PR[GP1:91,1] = PR[GP1:90,1] + 64.418;
   1:  PR[GP1:91,2] = PR[GP1:90,2] + 0.296;
   1:L PR[91] 10mm/sec CNT100;
   1:  PR[GP1:91,1] = PR[GP1:90,1] + 63.742;
   1:  PR[GP1:91,2] = PR[GP1:90,2] + 6.274;
   1:L PR[91] 10mm/sec CNT100;
   1:  PR[GP1:91,1] = PR[GP1:90,1] + 63.186;
   1:  PR[GP1:91,2] = PR[GP1:90,2] + 9.519;
   1:L PR[91] 10mm/sec CNT100;
   1:  PR[GP1:91,1] = PR[GP1:90,1] + 61.130;
   1:  PR[GP1:91,2] = PR[GP1:90,2] + 15.110;
   1:L PR[91] 10mm/sec CNT100;
   1:  PR[GP1:91,1] = PR[GP1:90,1] + 59.392;
   1:  PR[GP1:91,2] = PR[GP1:90,2] + 18.244;
   1:L PR[91] 10mm/sec CNT100;
   1:  PR[GP1:91,1] = PR[GP1:90,1] + 56.095;
   1:  PR[GP1:91,2] = PR[GP1:90,2] + 23.357;
   1:L PR[91] 10mm/sec CNT100;
   1:  PR[GP1:91,1] = PR[GP1:90,1] + 52.130;
   1:  PR[GP1:91,2] = PR[GP1:90,2] + 27.240;
   1:L PR[91] 10mm/sec CNT100;
   1:  PR[GP1:91,1] = PR[GP1:90,1] + 48.878;
   1:  PR[GP1:91,2] = PR[GP1:90,2] + 30.183;
   1:L PR[91] 10mm/sec CNT100;
   1:  PR[GP1:91,1] = PR[GP1:90,1] + 44.259;
   1:  PR[GP1:91,2] = PR[GP1:90,2] + 33.081;
   1:L PR[91] 10mm/sec CNT100;
   1:  PR[GP1:91,1] = PR[GP1:90,1] + 39.598;
   1:  PR[GP1:91,2] = PR[GP1:90,2] + 35.117;
   1:L PR[91] 10mm/sec CNT100;
   1:  PR[GP1:91,1] = PR[GP1:90,1] + 34.615;
   1:  PR[GP1:91,2] = PR[GP1:90,2] + 36.936;
   1:L PR[91] 10mm/sec CNT100;
   1:  PR[GP1:91,1] = PR[GP1:90,1] + 29.897;
   1:  PR[GP1:91,2] = PR[GP1:90,2] + 37.605;
   1:L PR[91] 10mm/sec CNT100;
   1:  PR[GP1:91,1] = PR[GP1:90,1] + 23.797;
   1:  PR[GP1:91,2] = PR[GP1:90,2] + 38.172;
   1:L PR[91] 10mm/sec CNT100;
   1:  PR[GP1:91,1] = PR[GP1:90,1] + 19.325;
   1:  PR[GP1:91,2] = PR[GP1:90,2] + 37.875;
   1:L PR[91] 10mm/sec CNT100;
   1:  PR[GP1:91,1] = PR[GP1:90,1] + 12.569;
   1:  PR[GP1:91,2] = PR[GP1:90,2] + 36.279;
   1:L PR[91] 10mm/sec CNT100;
   1:  PR[GP1:91,1] = PR[GP1:90,1] + 8.557;
   1:  PR[GP1:91,2] = PR[GP1:90,2] + 35.126;
   1:L PR[91] 10mm/sec CNT100;
   1:  PR[GP1:91,1] = PR[GP1:90,1] + 7.623;
   1:  PR[GP1:91,2] = PR[GP1:90,2] + 34.636;
   1:L PR[91] 10mm/sec CNT100;
   1:  PR[GP1:91,1] = PR[GP1:90,1] + 4.687;
   1:  PR[GP1:91,2] = PR[GP1:90,2] + 33.050;
   1:L PR[91] 10mm/sec CNT100;
   1:  PR[GP1:91,1] = PR[GP1:90,1] + -0.263;
   1:  PR[GP1:91,2] = PR[GP1:90,2] + 29.024;
   1:L PR[91] 10mm/sec CNT100;
   1:  PR[GP1:91,1] = PR[GP1:90,1] + -5.200;
   1:  PR[GP1:91,2] = PR[GP1:90,2] + 33.039;
   1:L PR[91] 10mm/sec CNT100;
   1:  PR[GP1:91,1] = PR[GP1:90,1] + -8.153;
   1:  PR[GP1:91,2] = PR[GP1:90,2] + 34.637;
   1:L PR[91] 10mm/sec CNT100;
   1:  PR[GP1:91,1] = PR[GP1:90,1] + -9.085;
   1:  PR[GP1:91,2] = PR[GP1:90,2] + 35.128;
   1:L PR[91] 10mm/sec CNT100;
   1:  PR[GP1:91,1] = PR[GP1:90,1] + -13.091;
   1:  PR[GP1:91,2] = PR[GP1:90,2] + 36.279;
   1:L PR[91] 10mm/sec CNT100;
   1:  PR[GP1:91,1] = PR[GP1:90,1] + -19.849;
   1:  PR[GP1:91,2] = PR[GP1:90,2] + 37.875;
   1:L PR[91] 10mm/sec CNT100;
   1:  PR[GP1:91,1] = PR[GP1:90,1] + -24.322;
   1:  PR[GP1:91,2] = PR[GP1:90,2] + 38.170;
   1:L PR[91] 10mm/sec CNT100;
   1:  PR[GP1:91,1] = PR[GP1:90,1] + -29.343;
   1:  PR[GP1:91,2] = PR[GP1:90,2] + 37.475;
   1:L PR[91] 10mm/sec CNT100;
   1:  PR[GP1:91,1] = PR[GP1:90,1] + -35.180;
   1:  PR[GP1:91,2] = PR[GP1:90,2] + 36.926;
   1:L PR[91] 10mm/sec CNT100;
   1:  PR[GP1:91,1] = PR[GP1:90,1] + -40.145;
   1:  PR[GP1:91,2] = PR[GP1:90,2] + 35.108;
   1:L PR[91] 10mm/sec CNT100;
   1:  PR[GP1:91,1] = PR[GP1:90,1] + -44.804;
   1:  PR[GP1:91,2] = PR[GP1:90,2] + 33.071;
   1:L PR[91] 10mm/sec CNT100;
   1:  PR[GP1:91,1] = PR[GP1:90,1] + -49.442;
   1:  PR[GP1:91,2] = PR[GP1:90,2] + 30.146;
   1:L PR[91] 10mm/sec CNT100;
   1:  PR[GP1:91,1] = PR[GP1:90,1] + -53.647;
   1:  PR[GP1:91,2] = PR[GP1:90,2] + 26.041;
   1:L PR[91] 10mm/sec CNT100;
   1:  PR[GP1:91,1] = PR[GP1:90,1] + -56.680;
   1:  PR[GP1:91,2] = PR[GP1:90,2] + 23.296;
   1:L PR[91] 10mm/sec CNT100;
   1:  PR[GP1:91,1] = PR[GP1:90,1] + -59.934;
   1:  PR[GP1:91,2] = PR[GP1:90,2] + 18.216;
   1:L PR[91] 10mm/sec CNT100;
   1:  PR[GP1:91,1] = PR[GP1:90,1] + -61.672;
   1:  PR[GP1:91,2] = PR[GP1:90,2] + 15.077;
   1:L PR[91] 10mm/sec CNT100;
   1:  PR[GP1:91,1] = PR[GP1:90,1] + -63.731;
   1:  PR[GP1:91,2] = PR[GP1:90,2] + 9.404;
   1:L PR[91] 10mm/sec CNT100;
   1:  PR[GP1:91,1] = PR[GP1:90,1] + -64.396;
   1:  PR[GP1:91,2] = PR[GP1:90,2] + 3.462;
   1:L PR[91] 10mm/sec CNT100;
   1:  PR[GP1:91,1] = PR[GP1:90,1] + -64.944;
   1:  PR[GP1:91,2] = PR[GP1:90,2] + 0.261;
   1:L PR[91] 10mm/sec CNT100;
   1:  PR[GP1:91,1] = PR[GP1:90,1] + -64.292;
   1:  PR[GP1:91,2] = PR[GP1:90,2] + -5.589;
   1:L PR[91] 10mm/sec CNT100;
   1:  PR[GP1:91,1] = PR[GP1:90,1] + -63.739;
   1:  PR[GP1:91,2] = PR[GP1:90,2] + -8.823;
   1:L PR[91] 10mm/sec CNT100;
   1:  PR[GP1:91,1] = PR[GP1:90,1] + -61.674;
   1:  PR[GP1:91,2] = PR[GP1:90,2] + -14.512;
   1:L PR[91] 10mm/sec CNT100;
   1:  PR[GP1:91,1] = PR[GP1:90,1] + -59.944;
   1:  PR[GP1:91,2] = PR[GP1:90,2] + -17.645;
   1:L PR[91] 10mm/sec CNT100;
   1:  PR[GP1:91,1] = PR[GP1:90,1] + -56.684;
   1:  PR[GP1:91,2] = PR[GP1:90,2] + -22.735;
   1:L PR[91] 10mm/sec CNT100;
   1:  PR[GP1:91,1] = PR[GP1:90,1] + -52.713;
   1:  PR[GP1:91,2] = PR[GP1:90,2] + -26.630;
   1:L PR[91] 10mm/sec CNT100;
   1:  PR[GP1:91,1] = PR[GP1:90,1] + -49.477;
   1:  PR[GP1:91,2] = PR[GP1:90,2] + -29.566;
   1:L PR[91] 10mm/sec CNT100;
   1:  PR[GP1:91,1] = PR[GP1:90,1] + -44.830;
   1:  PR[GP1:91,2] = PR[GP1:90,2] + -32.496;
   1:L PR[91] 10mm/sec CNT100;
   1:  PR[GP1:91,1] = PR[GP1:90,1] + -40.189;
   1:  PR[GP1:91,2] = PR[GP1:90,2] + -34.538;
   1:L PR[91] 10mm/sec CNT100;
   1:  PR[GP1:91,1] = PR[GP1:90,1] + -35.214;
   1:  PR[GP1:91,2] = PR[GP1:90,2] + -36.361;
   1:L PR[91] 10mm/sec CNT100;
   1:  PR[GP1:91,1] = PR[GP1:90,1] + -30.484;
   1:  PR[GP1:91,2] = PR[GP1:90,2] + -37.034;
   1:L PR[91] 10mm/sec CNT100;
   1:  PR[GP1:91,1] = PR[GP1:90,1] + -24.404;
   1:  PR[GP1:91,2] = PR[GP1:90,2] + -37.617;
   1:L PR[91] 10mm/sec CNT100;
   1:  PR[GP1:91,1] = PR[GP1:90,1] + -19.919;
   1:  PR[GP1:91,2] = PR[GP1:90,2] + -37.321;
   1:L PR[91] 10mm/sec CNT100;
   1:  PR[GP1:91,1] = PR[GP1:90,1] + -13.272;
   1:  PR[GP1:91,2] = PR[GP1:90,2] + -35.800;
   1:L PR[91] 10mm/sec CNT100;
   1:  PR[GP1:91,1] = PR[GP1:90,1] + -9.229;
   1:  PR[GP1:91,2] = PR[GP1:90,2] + -34.639;
   1:L PR[91] 10mm/sec CNT100;
   1:  PR[GP1:91,1] = PR[GP1:90,1] + -3.507;
   1:  PR[GP1:91,2] = PR[GP1:90,2] + -31.287;
   1:L PR[91] 10mm/sec CNT100;
   1:  PR[GP1:91,1] = PR[GP1:90,1] + -2.357;
   1:  PR[GP1:91,2] = PR[GP1:90,2] + -30.661;
   1:L PR[91] 10mm/sec CNT100;
   1:  PR[GP1:91,1] = PR[GP1:90,1] + -0.265;
   1:  PR[GP1:91,2] = PR[GP1:90,2] + -28.855;
   1:L PR[91] 10mm/sec CNT100;
   1:  PR[GP1:91,1] = PR[GP1:90,1] + 1.586;
   1:  PR[GP1:91,2] = PR[GP1:90,2] + -30.734;
   1:  PR[GP1:91,3] = PR[GP1:90,3] + 64.355;
   1:L PR[91] 10mm/sec CNT100;
   1:  PR[GP1:91,1] = PR[GP1:90,1] + 2.563;
   1:  PR[GP1:91,2] = PR[GP1:90,2] + -31.264;
   1:L PR[91] 10mm/sec CNT100;
   1:  PR[GP1:91,1] = PR[GP1:90,1] + 8.444;
   1:  PR[GP1:91,2] = PR[GP1:90,2] + -34.707;
   1:L PR[91] 10mm/sec CNT100;
   1:  PR[GP1:91,1] = PR[GP1:90,1] + 12.372;
   1:  PR[GP1:91,2] = PR[GP1:90,2] + -35.835;
   1:L PR[91] 10mm/sec CNT100;
   1:  PR[GP1:91,1] = PR[GP1:90,1] + 19.217;
   1:  PR[GP1:91,2] = PR[GP1:90,2] + -37.401;
   1:L PR[91] 10mm/sec CNT100;
   1:  PR[GP1:91,1] = PR[GP1:90,1] + 23.553;
   1:  PR[GP1:91,2] = PR[GP1:90,2] + -37.689;
   1:L PR[91] 10mm/sec CNT100;
   1:  PR[GP1:91,1] = PR[GP1:90,1] + 28.419;
   1:  PR[GP1:91,2] = PR[GP1:90,2] + -37.017;
   1:L PR[91] 10mm/sec CNT100;
   1:  PR[GP1:91,1] = PR[GP1:90,1] + 34.457;
   1:  PR[GP1:91,2] = PR[GP1:90,2] + -36.431;
   1:L PR[91] 10mm/sec CNT100;
   1:  PR[GP1:91,1] = PR[GP1:90,1] + 39.298;
   1:  PR[GP1:91,2] = PR[GP1:90,2] + -34.664;
   1:L PR[91] 10mm/sec CNT100;
   1:  PR[GP1:91,1] = PR[GP1:90,1] + 44.140;
   1:  PR[GP1:91,2] = PR[GP1:90,2] + -32.534;
   1:L PR[91] 10mm/sec CNT100;
   1:  PR[GP1:91,1] = PR[GP1:90,1] + 48.638;
   1:  PR[GP1:91,2] = PR[GP1:90,2] + -29.712;
   1:L PR[91] 10mm/sec CNT100;
   1:  PR[GP1:91,1] = PR[GP1:90,1] + 52.734;
   1:  PR[GP1:91,2] = PR[GP1:90,2] + -25.720;
   1:L PR[91] 10mm/sec CNT100;
   1:  PR[GP1:91,1] = PR[GP1:90,1] + 55.925;
   1:  PR[GP1:91,2] = PR[GP1:90,2] + -22.817;
   1:L PR[91] 10mm/sec CNT100;
   1:  PR[GP1:91,1] = PR[GP1:90,1] + 59.140;
   1:  PR[GP1:91,2] = PR[GP1:90,2] + -17.831;
   1:L PR[91] 10mm/sec CNT100;
   1:  PR[GP1:91,1] = PR[GP1:90,1] + 60.978;
   1:  PR[GP1:91,2] = PR[GP1:90,2] + -14.508;
   1:L PR[91] 10mm/sec CNT100;
   1:  PR[GP1:91,1] = PR[GP1:90,1] + 62.983;
   1:  PR[GP1:91,2] = PR[GP1:90,2] + -9.057;
   1:L PR[91] 10mm/sec CNT100;
   1:  PR[GP1:91,1] = PR[GP1:90,1] + 63.658;
   1:  PR[GP1:91,2] = PR[GP1:90,2] + -3.120;
   1:L PR[91] 10mm/sec CNT100;
   1:  PR[GP1:91,1] = PR[GP1:90,1] + 64.240;
   1:  PR[GP1:91,2] = PR[GP1:90,2] + 0.296;
   1:L PR[91] 10mm/sec CNT100;
   1:  PR[GP1:91,1] = PR[GP1:90,1] + 63.579;
   1:  PR[GP1:91,2] = PR[GP1:90,2] + 6.143;
   1:L PR[91] 10mm/sec CNT100;
   1:  PR[GP1:91,1] = PR[GP1:90,1] + 62.986;
   1:  PR[GP1:91,2] = PR[GP1:90,2] + 9.607;
   1:L PR[91] 10mm/sec CNT100;
   1:  PR[GP1:91,1] = PR[GP1:90,1] + 60.976;
   1:  PR[GP1:91,2] = PR[GP1:90,2] + 15.074;
   1:L PR[91] 10mm/sec CNT100;
   1:  PR[GP1:91,1] = PR[GP1:90,1] + 59.129;
   1:  PR[GP1:91,2] = PR[GP1:90,2] + 18.403;
   1:L PR[91] 10mm/sec CNT100;
   1:  PR[GP1:91,1] = PR[GP1:90,1] + 55.908;
   1:  PR[GP1:91,2] = PR[GP1:90,2] + 23.399;
   1:L PR[91] 10mm/sec CNT100;
   1:  PR[GP1:91,1] = PR[GP1:90,1] + 52.033;
   1:  PR[GP1:91,2] = PR[GP1:90,2] + 27.194;
   1:L PR[91] 10mm/sec CNT100;
   1:  PR[GP1:91,1] = PR[GP1:90,1] + 48.622;
   1:  PR[GP1:91,2] = PR[GP1:90,2] + 30.281;
   1:L PR[91] 10mm/sec CNT100;
   1:  PR[GP1:91,1] = PR[GP1:90,1] + 44.113;
   1:  PR[GP1:91,2] = PR[GP1:90,2] + 33.110;
   1:L PR[91] 10mm/sec CNT100;
   1:  PR[GP1:91,1] = PR[GP1:90,1] + 39.252;
   1:  PR[GP1:91,2] = PR[GP1:90,2] + 35.234;
   1:L PR[91] 10mm/sec CNT100;
   1:  PR[GP1:91,1] = PR[GP1:90,1] + 34.395;
   1:  PR[GP1:91,2] = PR[GP1:90,2] + 37.006;
   1:L PR[91] 10mm/sec CNT100;
   1:  PR[GP1:91,1] = PR[GP1:90,1] + 29.798;
   1:  PR[GP1:91,2] = PR[GP1:90,2] + 37.658;
   1:L PR[91] 10mm/sec CNT100;
   1:  PR[GP1:91,1] = PR[GP1:90,1] + 23.495;
   1:  PR[GP1:91,2] = PR[GP1:90,2] + 38.244;
   1:L PR[91] 10mm/sec CNT100;
   1:  PR[GP1:91,1] = PR[GP1:90,1] + 19.146;
   1:  PR[GP1:91,2] = PR[GP1:90,2] + 37.955;
   1:L PR[91] 10mm/sec CNT100;
   1:  PR[GP1:91,1] = PR[GP1:90,1] + 12.188;
   1:  PR[GP1:91,2] = PR[GP1:90,2] + 36.311;
   1:L PR[91] 10mm/sec CNT100;
   1:  PR[GP1:91,1] = PR[GP1:90,1] + 8.299;
   1:  PR[GP1:91,2] = PR[GP1:90,2] + 35.193;
   1:L PR[91] 10mm/sec CNT100;
   1:  PR[GP1:91,1] = PR[GP1:90,1] + 7.339;
   1:  PR[GP1:91,2] = PR[GP1:90,2] + 34.690;
   1:L PR[91] 10mm/sec CNT100;
   1:  PR[GP1:91,1] = PR[GP1:90,1] + 4.514;
   1:  PR[GP1:91,2] = PR[GP1:90,2] + 33.165;
   1:L PR[91] 10mm/sec CNT100;
   1:  PR[GP1:91,1] = PR[GP1:90,1] + -0.263;
   1:  PR[GP1:91,2] = PR[GP1:90,2] + 29.279;
   1:L PR[91] 10mm/sec CNT100;
   1:  PR[GP1:91,1] = PR[GP1:90,1] + -5.028;
   1:  PR[GP1:91,2] = PR[GP1:90,2] + 33.153;
   1:L PR[91] 10mm/sec CNT100;
   1:  PR[GP1:91,1] = PR[GP1:90,1] + -7.869;
   1:  PR[GP1:91,2] = PR[GP1:90,2] + 34.691;
   1:L PR[91] 10mm/sec CNT100;
   1:  PR[GP1:91,1] = PR[GP1:90,1] + -8.827;
   1:  PR[GP1:91,2] = PR[GP1:90,2] + 35.195;
   1:L PR[91] 10mm/sec CNT100;
   1:  PR[GP1:91,1] = PR[GP1:90,1] + -12.710;
   1:  PR[GP1:91,2] = PR[GP1:90,2] + 36.312;
   1:L PR[91] 10mm/sec CNT100;
   1:  PR[GP1:91,1] = PR[GP1:90,1] + -19.670;
   1:  PR[GP1:91,2] = PR[GP1:90,2] + 37.955;
   1:L PR[91] 10mm/sec CNT100;
   1:  PR[GP1:91,1] = PR[GP1:90,1] + -24.019;
   1:  PR[GP1:91,2] = PR[GP1:90,2] + 38.242;
   1:L PR[91] 10mm/sec CNT100;
   1:  PR[GP1:91,1] = PR[GP1:90,1] + -28.904;
   1:  PR[GP1:91,2] = PR[GP1:90,2] + 37.566;
   1:L PR[91] 10mm/sec CNT100;
   1:  PR[GP1:91,1] = PR[GP1:90,1] + -34.961;
   1:  PR[GP1:91,2] = PR[GP1:90,2] + 36.996;
   1:L PR[91] 10mm/sec CNT100;
   1:  PR[GP1:91,1] = PR[GP1:90,1] + -39.798;
   1:  PR[GP1:91,2] = PR[GP1:90,2] + 35.225;
   1:L PR[91] 10mm/sec CNT100;
   1:  PR[GP1:91,1] = PR[GP1:90,1] + -44.657;
   1:  PR[GP1:91,2] = PR[GP1:90,2] + 33.100;
   1:L PR[91] 10mm/sec CNT100;
   1:  PR[GP1:91,1] = PR[GP1:90,1] + -49.184;
   1:  PR[GP1:91,2] = PR[GP1:90,2] + 30.246;
   1:L PR[91] 10mm/sec CNT100;
   1:  PR[GP1:91,1] = PR[GP1:90,1] + -53.290;
   1:  PR[GP1:91,2] = PR[GP1:90,2] + 26.238;
   1:L PR[91] 10mm/sec CNT100;
   1:  PR[GP1:91,1] = PR[GP1:90,1] + -56.491;
   1:  PR[GP1:91,2] = PR[GP1:90,2] + 23.339;
   1:L PR[91] 10mm/sec CNT100;
   1:  PR[GP1:91,1] = PR[GP1:90,1] + -59.671;
   1:  PR[GP1:91,2] = PR[GP1:90,2] + 18.375;
   1:L PR[91] 10mm/sec CNT100;
   1:  PR[GP1:91,1] = PR[GP1:90,1] + -61.517;
   1:  PR[GP1:91,2] = PR[GP1:90,2] + 15.041;
   1:L PR[91] 10mm/sec CNT100;
   1:  PR[GP1:91,1] = PR[GP1:90,1] + -63.531;
   1:  PR[GP1:91,2] = PR[GP1:90,2] + 9.494;
   1:L PR[91] 10mm/sec CNT100;
   1:  PR[GP1:91,1] = PR[GP1:90,1] + -64.182;
   1:  PR[GP1:91,2] = PR[GP1:90,2] + 3.682;
   1:L PR[91] 10mm/sec CNT100;
   1:  PR[GP1:91,1] = PR[GP1:90,1] + -64.767;
   1:  PR[GP1:91,2] = PR[GP1:90,2] + 0.261;
   1:L PR[91] 10mm/sec CNT100;
   1:  PR[GP1:91,1] = PR[GP1:90,1] + -64.129;
   1:  PR[GP1:91,2] = PR[GP1:90,2] + -5.461;
   1:L PR[91] 10mm/sec CNT100;
   1:  PR[GP1:91,1] = PR[GP1:90,1] + -63.539;
   1:  PR[GP1:91,2] = PR[GP1:90,2] + -8.912;
   1:L PR[91] 10mm/sec CNT100;
   1:  PR[GP1:91,1] = PR[GP1:90,1] + -61.520;
   1:  PR[GP1:91,2] = PR[GP1:90,2] + -14.476;
   1:L PR[91] 10mm/sec CNT100;
   1:  PR[GP1:91,1] = PR[GP1:90,1] + -59.682;
   1:  PR[GP1:91,2] = PR[GP1:90,2] + -17.804;
   1:L PR[91] 10mm/sec CNT100;
   1:  PR[GP1:91,1] = PR[GP1:90,1] + -56.496;
   1:  PR[GP1:91,2] = PR[GP1:90,2] + -22.777;
   1:L PR[91] 10mm/sec CNT100;
   1:  PR[GP1:91,1] = PR[GP1:90,1] + -52.615;
   1:  PR[GP1:91,2] = PR[GP1:90,2] + -26.585;
   1:L PR[91] 10mm/sec CNT100;
   1:  PR[GP1:91,1] = PR[GP1:90,1] + -49.220;
   1:  PR[GP1:91,2] = PR[GP1:90,2] + -29.665;
   1:L PR[91] 10mm/sec CNT100;
   1:  PR[GP1:91,1] = PR[GP1:90,1] + -44.685;
   1:  PR[GP1:91,2] = PR[GP1:90,2] + -32.524;
   1:L PR[91] 10mm/sec CNT100;
   1:  PR[GP1:91,1] = PR[GP1:90,1] + -39.844;
   1:  PR[GP1:91,2] = PR[GP1:90,2] + -34.654;
   1:L PR[91] 10mm/sec CNT100;
   1:  PR[GP1:91,1] = PR[GP1:90,1] + -34.996;
   1:  PR[GP1:91,2] = PR[GP1:90,2] + -36.430;
   1:L PR[91] 10mm/sec CNT100;
   1:  PR[GP1:91,1] = PR[GP1:90,1] + -30.386;
   1:  PR[GP1:91,2] = PR[GP1:90,2] + -37.086;
   1:L PR[91] 10mm/sec CNT100;
   1:  PR[GP1:91,1] = PR[GP1:90,1] + -24.104;
   1:  PR[GP1:91,2] = PR[GP1:90,2] + -37.689;
   1:L PR[91] 10mm/sec CNT100;
   1:  PR[GP1:91,1] = PR[GP1:90,1] + -19.742;
   1:  PR[GP1:91,2] = PR[GP1:90,2] + -37.401;
   1:L PR[91] 10mm/sec CNT100;
   1:  PR[GP1:91,1] = PR[GP1:90,1] + -12.897;
   1:  PR[GP1:91,2] = PR[GP1:90,2] + -35.835;
   1:L PR[91] 10mm/sec CNT100;
   1:  PR[GP1:91,1] = PR[GP1:90,1] + -8.974;
   1:  PR[GP1:91,2] = PR[GP1:90,2] + -34.709;
   1:L PR[91] 10mm/sec CNT100;
   1:  PR[GP1:91,1] = PR[GP1:90,1] + -3.097;
   1:  PR[GP1:91,2] = PR[GP1:90,2] + -31.265;
   1:L PR[91] 10mm/sec CNT100;
   1:  PR[GP1:91,1] = PR[GP1:90,1] + -2.114;
   1:  PR[GP1:91,2] = PR[GP1:90,2] + -30.730;
   1:L PR[91] 10mm/sec CNT100;
   1:  PR[GP1:91,1] = PR[GP1:90,1] + -0.265;
   1:  PR[GP1:91,2] = PR[GP1:90,2] + -29.135;
   1:L PR[91] 10mm/sec CNT100;
   1:  PR[GP1:91,1] = PR[GP1:90,1] + 1.341;
   1:  PR[GP1:91,2] = PR[GP1:90,2] + -30.802;
   1:  PR[GP1:91,3] = PR[GP1:90,3] + 64.965;
   1:L PR[91] 10mm/sec CNT100;
   1:  PR[GP1:91,1] = PR[GP1:90,1] + 2.152;
   1:  PR[GP1:91,2] = PR[GP1:90,2] + -31.243;
   1:L PR[91] 10mm/sec CNT100;
   1:  PR[GP1:91,1] = PR[GP1:90,1] + 8.189;
   1:  PR[GP1:91,2] = PR[GP1:90,2] + -34.776;
   1:L PR[91] 10mm/sec CNT100;
   1:  PR[GP1:91,1] = PR[GP1:90,1] + 11.997;
   1:  PR[GP1:91,2] = PR[GP1:90,2] + -35.870;
   1:L PR[91] 10mm/sec CNT100;
   1:  PR[GP1:91,1] = PR[GP1:90,1] + 19.040;
   1:  PR[GP1:91,2] = PR[GP1:90,2] + -37.481;
   1:L PR[91] 10mm/sec CNT100;
   1:  PR[GP1:91,1] = PR[GP1:90,1] + 23.253;
   1:  PR[GP1:91,2] = PR[GP1:90,2] + -37.761;
   1:L PR[91] 10mm/sec CNT100;
   1:  PR[GP1:91,1] = PR[GP1:90,1] + 27.982;
   1:  PR[GP1:91,2] = PR[GP1:90,2] + -37.108;
   1:L PR[91] 10mm/sec CNT100;
   1:  PR[GP1:91,1] = PR[GP1:90,1] + 34.239;
   1:  PR[GP1:91,2] = PR[GP1:90,2] + -36.500;
   1:L PR[91] 10mm/sec CNT100;
   1:  PR[GP1:91,1] = PR[GP1:90,1] + 38.954;
   1:  PR[GP1:91,2] = PR[GP1:90,2] + -34.779;
   1:L PR[91] 10mm/sec CNT100;
   1:  PR[GP1:91,1] = PR[GP1:90,1] + 43.995;
   1:  PR[GP1:91,2] = PR[GP1:90,2] + -32.563;
   1:L PR[91] 10mm/sec CNT100;
   1:  PR[GP1:91,1] = PR[GP1:90,1] + 48.383;
   1:  PR[GP1:91,2] = PR[GP1:90,2] + -29.810;
   1:L PR[91] 10mm/sec CNT100;
   1:  PR[GP1:91,1] = PR[GP1:90,1] + 52.379;
   1:  PR[GP1:91,2] = PR[GP1:90,2] + -25.914;
   1:L PR[91] 10mm/sec CNT100;
   1:  PR[GP1:91,1] = PR[GP1:90,1] + 55.738;
   1:  PR[GP1:91,2] = PR[GP1:90,2] + -22.859;
   1:L PR[91] 10mm/sec CNT100;
   1:  PR[GP1:91,1] = PR[GP1:90,1] + 58.878;
   1:  PR[GP1:91,2] = PR[GP1:90,2] + -17.989;
   1:L PR[91] 10mm/sec CNT100;
   1:  PR[GP1:91,1] = PR[GP1:90,1] + 60.824;
   1:  PR[GP1:91,2] = PR[GP1:90,2] + -14.472;
   1:L PR[91] 10mm/sec CNT100;
   1:  PR[GP1:91,1] = PR[GP1:90,1] + 62.783;
   1:  PR[GP1:91,2] = PR[GP1:90,2] + -9.144;
   1:L PR[91] 10mm/sec CNT100;
   1:  PR[GP1:91,1] = PR[GP1:90,1] + 63.443;
   1:  PR[GP1:91,2] = PR[GP1:90,2] + -3.340;
   1:L PR[91] 10mm/sec CNT100;
   1:  PR[GP1:91,1] = PR[GP1:90,1] + 64.063;
   1:  PR[GP1:91,2] = PR[GP1:90,2] + 0.296;
   1:L PR[91] 10mm/sec CNT100;
   1:  PR[GP1:91,1] = PR[GP1:90,1] + 63.417;
   1:  PR[GP1:91,2] = PR[GP1:90,2] + 6.013;
   1:L PR[91] 10mm/sec CNT100;
   1:  PR[GP1:91,1] = PR[GP1:90,1] + 62.787;
   1:  PR[GP1:91,2] = PR[GP1:90,2] + 9.694;
   1:L PR[91] 10mm/sec CNT100;
   1:  PR[GP1:91,1] = PR[GP1:90,1] + 60.821;
   1:  PR[GP1:91,2] = PR[GP1:90,2] + 15.037;
   1:L PR[91] 10mm/sec CNT100;
   1:  PR[GP1:91,1] = PR[GP1:90,1] + 58.867;
   1:  PR[GP1:91,2] = PR[GP1:90,2] + 18.561;
   1:L PR[91] 10mm/sec CNT100;
   1:  PR[GP1:91,1] = PR[GP1:90,1] + 55.720;
   1:  PR[GP1:91,2] = PR[GP1:90,2] + 23.441;
   1:L PR[91] 10mm/sec CNT100;
   1:  PR[GP1:91,1] = PR[GP1:90,1] + 51.935;
   1:  PR[GP1:91,2] = PR[GP1:90,2] + 27.148;
   1:L PR[91] 10mm/sec CNT100;
   1:  PR[GP1:91,1] = PR[GP1:90,1] + 48.365;
   1:  PR[GP1:91,2] = PR[GP1:90,2] + 30.379;
   1:L PR[91] 10mm/sec CNT100;
   1:  PR[GP1:91,1] = PR[GP1:90,1] + 43.966;
   1:  PR[GP1:91,2] = PR[GP1:90,2] + 33.139;
   1:L PR[91] 10mm/sec CNT100;
   1:  PR[GP1:91,1] = PR[GP1:90,1] + 38.906;
   1:  PR[GP1:91,2] = PR[GP1:90,2] + 35.350;
   1:L PR[91] 10mm/sec CNT100;
   1:  PR[GP1:91,1] = PR[GP1:90,1] + 34.176;
   1:  PR[GP1:91,2] = PR[GP1:90,2] + 37.076;
   1:L PR[91] 10mm/sec CNT100;
   1:  PR[GP1:91,1] = PR[GP1:90,1] + 29.699;
   1:  PR[GP1:91,2] = PR[GP1:90,2] + 37.711;
   1:L PR[91] 10mm/sec CNT100;
   1:  PR[GP1:91,1] = PR[GP1:90,1] + 23.193;
   1:  PR[GP1:91,2] = PR[GP1:90,2] + 38.315;
   1:L PR[91] 10mm/sec CNT100;
   1:  PR[GP1:91,1] = PR[GP1:90,1] + 18.967;
   1:  PR[GP1:91,2] = PR[GP1:90,2] + 38.035;
   1:L PR[91] 10mm/sec CNT100;
   1:  PR[GP1:91,1] = PR[GP1:90,1] + 11.807;
   1:  PR[GP1:91,2] = PR[GP1:90,2] + 36.344;
   1:L PR[91] 10mm/sec CNT100;
   1:  PR[GP1:91,1] = PR[GP1:90,1] + 8.041;
   1:  PR[GP1:91,2] = PR[GP1:90,2] + 35.261;
   1:L PR[91] 10mm/sec CNT100;
   1:  PR[GP1:91,1] = PR[GP1:90,1] + 7.054;
   1:  PR[GP1:91,2] = PR[GP1:90,2] + 34.743;
   1:L PR[91] 10mm/sec CNT100;
   1:  PR[GP1:91,1] = PR[GP1:90,1] + 4.341;
   1:  PR[GP1:91,2] = PR[GP1:90,2] + 33.279;
   1:L PR[91] 10mm/sec CNT100;
   1:  PR[GP1:91,1] = PR[GP1:90,1] + -0.263;
   1:  PR[GP1:91,2] = PR[GP1:90,2] + 29.534;
   1:L PR[91] 10mm/sec CNT100;
   1:  PR[GP1:91,1] = PR[GP1:90,1] + -4.856;
   1:  PR[GP1:91,2] = PR[GP1:90,2] + 33.268;
   1:L PR[91] 10mm/sec CNT100;
   1:  PR[GP1:91,1] = PR[GP1:90,1] + -7.584;
   1:  PR[GP1:91,2] = PR[GP1:90,2] + 34.745;
   1:L PR[91] 10mm/sec CNT100;
   1:  PR[GP1:91,1] = PR[GP1:90,1] + -8.569;
   1:  PR[GP1:91,2] = PR[GP1:90,2] + 35.263;
   1:L PR[91] 10mm/sec CNT100;
   1:  PR[GP1:91,1] = PR[GP1:90,1] + -12.329;
   1:  PR[GP1:91,2] = PR[GP1:90,2] + 36.344;
   1:L PR[91] 10mm/sec CNT100;
   1:  PR[GP1:91,1] = PR[GP1:90,1] + -19.491;
   1:  PR[GP1:91,2] = PR[GP1:90,2] + 38.035;
   1:L PR[91] 10mm/sec CNT100;
   1:  PR[GP1:91,1] = PR[GP1:90,1] + -23.717;
   1:  PR[GP1:91,2] = PR[GP1:90,2] + 38.314;
   1:L PR[91] 10mm/sec CNT100;
   1:  PR[GP1:91,1] = PR[GP1:90,1] + -28.465;
   1:  PR[GP1:91,2] = PR[GP1:90,2] + 37.657;
   1:L PR[91] 10mm/sec CNT100;
   1:  PR[GP1:91,1] = PR[GP1:90,1] + -34.741;
   1:  PR[GP1:91,2] = PR[GP1:90,2] + 37.067;
   1:L PR[91] 10mm/sec CNT100;
   1:  PR[GP1:91,1] = PR[GP1:90,1] + -39.452;
   1:  PR[GP1:91,2] = PR[GP1:90,2] + 35.341;
   1:L PR[91] 10mm/sec CNT100;
   1:  PR[GP1:91,1] = PR[GP1:90,1] + -44.510;
   1:  PR[GP1:91,2] = PR[GP1:90,2] + 33.129;
   1:L PR[91] 10mm/sec CNT100;
   1:  PR[GP1:91,1] = PR[GP1:90,1] + -48.926;
   1:  PR[GP1:91,2] = PR[GP1:90,2] + 30.345;
   1:L PR[91] 10mm/sec CNT100;
   1:  PR[GP1:91,1] = PR[GP1:90,1] + -52.932;
   1:  PR[GP1:91,2] = PR[GP1:90,2] + 26.434;
   1:L PR[91] 10mm/sec CNT100;
   1:  PR[GP1:91,1] = PR[GP1:90,1] + -56.302;
   1:  PR[GP1:91,2] = PR[GP1:90,2] + 23.383;
   1:L PR[91] 10mm/sec CNT100;
   1:  PR[GP1:91,1] = PR[GP1:90,1] + -59.409;
   1:  PR[GP1:91,2] = PR[GP1:90,2] + 18.534;
   1:L PR[91] 10mm/sec CNT100;
   1:  PR[GP1:91,1] = PR[GP1:90,1] + -61.362;
   1:  PR[GP1:91,2] = PR[GP1:90,2] + 15.005;
   1:L PR[91] 10mm/sec CNT100;
   1:  PR[GP1:91,1] = PR[GP1:90,1] + -63.330;
   1:  PR[GP1:91,2] = PR[GP1:90,2] + 9.584;
   1:L PR[91] 10mm/sec CNT100;
   1:  PR[GP1:91,1] = PR[GP1:90,1] + -63.967;
   1:  PR[GP1:91,2] = PR[GP1:90,2] + 3.902;
   1:L PR[91] 10mm/sec CNT100;
   1:  PR[GP1:91,1] = PR[GP1:90,1] + -64.590;
   1:  PR[GP1:91,2] = PR[GP1:90,2] + 0.261;
   1:L PR[91] 10mm/sec CNT100;
   1:  PR[GP1:91,1] = PR[GP1:90,1] + -63.966;
   1:  PR[GP1:91,2] = PR[GP1:90,2] + -5.333;
   1:L PR[91] 10mm/sec CNT100;
   1:  PR[GP1:91,1] = PR[GP1:90,1] + -63.339;
   1:  PR[GP1:91,2] = PR[GP1:90,2] + -9.002;
   1:L PR[91] 10mm/sec CNT100;
   1:  PR[GP1:91,1] = PR[GP1:90,1] + -61.365;
   1:  PR[GP1:91,2] = PR[GP1:90,2] + -14.440;
   1:L PR[91] 10mm/sec CNT100;
   1:  PR[GP1:91,1] = PR[GP1:90,1] + -59.420;
   1:  PR[GP1:91,2] = PR[GP1:90,2] + -17.962;
   1:L PR[91] 10mm/sec CNT100;
   1:  PR[GP1:91,1] = PR[GP1:90,1] + -56.308;
   1:  PR[GP1:91,2] = PR[GP1:90,2] + -22.820;
   1:L PR[91] 10mm/sec CNT100;
   1:  PR[GP1:91,1] = PR[GP1:90,1] + -52.517;
   1:  PR[GP1:91,2] = PR[GP1:90,2] + -26.539;
   1:L PR[91] 10mm/sec CNT100;
   1:  PR[GP1:91,1] = PR[GP1:90,1] + -48.963;
   1:  PR[GP1:91,2] = PR[GP1:90,2] + -29.763;
   1:L PR[91] 10mm/sec CNT100;
   1:  PR[GP1:91,1] = PR[GP1:90,1] + -44.539;
   1:  PR[GP1:91,2] = PR[GP1:90,2] + -32.553;
   1:L PR[91] 10mm/sec CNT100;
   1:  PR[GP1:91,1] = PR[GP1:90,1] + -39.500;
   1:  PR[GP1:91,2] = PR[GP1:90,2] + -34.770;
   1:L PR[91] 10mm/sec CNT100;
   1:  PR[GP1:91,1] = PR[GP1:90,1] + -34.778;
   1:  PR[GP1:91,2] = PR[GP1:90,2] + -36.500;
   1:L PR[91] 10mm/sec CNT100;
   1:  PR[GP1:91,1] = PR[GP1:90,1] + -30.288;
   1:  PR[GP1:91,2] = PR[GP1:90,2] + -37.139;
   1:L PR[91] 10mm/sec CNT100;
   1:  PR[GP1:91,1] = PR[GP1:90,1] + -23.803;
   1:  PR[GP1:91,2] = PR[GP1:90,2] + -37.761;
   1:L PR[91] 10mm/sec CNT100;
   1:  PR[GP1:91,1] = PR[GP1:90,1] + -19.565;
   1:  PR[GP1:91,2] = PR[GP1:90,2] + -37.481;
   1:L PR[91] 10mm/sec CNT100;
   1:  PR[GP1:91,1] = PR[GP1:90,1] + -12.521;
   1:  PR[GP1:91,2] = PR[GP1:90,2] + -35.870;
   1:L PR[91] 10mm/sec CNT100;
   1:  PR[GP1:91,1] = PR[GP1:90,1] + -8.720;
   1:  PR[GP1:91,2] = PR[GP1:90,2] + -34.778;
   1:L PR[91] 10mm/sec CNT100;
   1:  PR[GP1:91,1] = PR[GP1:90,1] + -2.686;
   1:  PR[GP1:91,2] = PR[GP1:90,2] + -31.243;
   1:L PR[91] 10mm/sec CNT100;
   1:  PR[GP1:91,1] = PR[GP1:90,1] + -1.870;
   1:  PR[GP1:91,2] = PR[GP1:90,2] + -30.799;
   1:L PR[91] 10mm/sec CNT100;
   1:  PR[GP1:91,1] = PR[GP1:90,1] + -0.265;
   1:  PR[GP1:91,2] = PR[GP1:90,2] + -29.414;
   1:L PR[91] 10mm/sec CNT100;
   1:  PR[GP1:91,1] = PR[GP1:90,1] + 1.097;
   1:  PR[GP1:91,2] = PR[GP1:90,2] + -30.871;
   1:  PR[GP1:91,3] = PR[GP1:90,3] + 65.575;
   1:L PR[91] 10mm/sec CNT100;
   1:  PR[GP1:91,1] = PR[GP1:90,1] + 1.742;
   1:  PR[GP1:91,2] = PR[GP1:90,2] + -31.221;
   1:L PR[91] 10mm/sec CNT100;
   1:  PR[GP1:91,1] = PR[GP1:90,1] + 7.935;
   1:  PR[GP1:91,2] = PR[GP1:90,2] + -34.846;
   1:L PR[91] 10mm/sec CNT100;
   1:  PR[GP1:91,1] = PR[GP1:90,1] + 11.621;
   1:  PR[GP1:91,2] = PR[GP1:90,2] + -35.904;
   1:L PR[91] 10mm/sec CNT100;
   1:  PR[GP1:91,1] = PR[GP1:90,1] + 18.863;
   1:  PR[GP1:91,2] = PR[GP1:90,2] + -37.562;
   1:L PR[91] 10mm/sec CNT100;
   1:  PR[GP1:91,1] = PR[GP1:90,1] + 22.953;
   1:  PR[GP1:91,2] = PR[GP1:90,2] + -37.833;
   1:L PR[91] 10mm/sec CNT100;
   1:  PR[GP1:91,1] = PR[GP1:90,1] + 27.546;
   1:  PR[GP1:91,2] = PR[GP1:90,2] + -37.199;
   1:L PR[91] 10mm/sec CNT100;
   1:  PR[GP1:91,1] = PR[GP1:90,1] + 34.022;
   1:  PR[GP1:91,2] = PR[GP1:90,2] + -36.570;
   1:L PR[91] 10mm/sec CNT100;
   1:  PR[GP1:91,1] = PR[GP1:90,1] + 38.610;
   1:  PR[GP1:91,2] = PR[GP1:90,2] + -34.895;
   1:L PR[91] 10mm/sec CNT100;
   1:  PR[GP1:91,1] = PR[GP1:90,1] + 43.850;
   1:  PR[GP1:91,2] = PR[GP1:90,2] + -32.591;
   1:L PR[91] 10mm/sec CNT100;
   1:  PR[GP1:91,1] = PR[GP1:90,1] + 48.127;
   1:  PR[GP1:91,2] = PR[GP1:90,2] + -29.907;
   1:L PR[91] 10mm/sec CNT100;
   1:  PR[GP1:91,1] = PR[GP1:90,1] + 52.024;
   1:  PR[GP1:91,2] = PR[GP1:90,2] + -26.109;
   1:L PR[91] 10mm/sec CNT100;
   1:  PR[GP1:91,1] = PR[GP1:90,1] + 55.552;
   1:  PR[GP1:91,2] = PR[GP1:90,2] + -22.900;
   1:L PR[91] 10mm/sec CNT100;
   1:  PR[GP1:91,1] = PR[GP1:90,1] + 58.616;
   1:  PR[GP1:91,2] = PR[GP1:90,2] + -18.147;
   1:L PR[91] 10mm/sec CNT100;
   1:  PR[GP1:91,1] = PR[GP1:90,1] + 60.670;
   1:  PR[GP1:91,2] = PR[GP1:90,2] + -14.435;
   1:L PR[91] 10mm/sec CNT100;
   1:  PR[GP1:91,1] = PR[GP1:90,1] + 62.584;
   1:  PR[GP1:91,2] = PR[GP1:90,2] + -9.231;
   1:L PR[91] 10mm/sec CNT100;
   1:  PR[GP1:91,1] = PR[GP1:90,1] + 63.228;
   1:  PR[GP1:91,2] = PR[GP1:90,2] + -3.560;
   1:L PR[91] 10mm/sec CNT100;
   1:  PR[GP1:91,1] = PR[GP1:90,1] + 63.886;
   1:  PR[GP1:91,2] = PR[GP1:90,2] + 0.296;
   1:L PR[91] 10mm/sec CNT100;
   1:  PR[GP1:91,1] = PR[GP1:90,1] + 63.254;
   1:  PR[GP1:91,2] = PR[GP1:90,2] + 5.882;
   1:L PR[91] 10mm/sec CNT100;
   1:  PR[GP1:91,1] = PR[GP1:90,1] + 62.587;
   1:  PR[GP1:91,2] = PR[GP1:90,2] + 9.781;
   1:L PR[91] 10mm/sec CNT100;
   1:  PR[GP1:91,1] = PR[GP1:90,1] + 60.667;
   1:  PR[GP1:91,2] = PR[GP1:90,2] + 15.001;
   1:L PR[91] 10mm/sec CNT100;
   1:  PR[GP1:91,1] = PR[GP1:90,1] + 58.605;
   1:  PR[GP1:91,2] = PR[GP1:90,2] + 18.719;
   1:L PR[91] 10mm/sec CNT100;
   1:  PR[GP1:91,1] = PR[GP1:90,1] + 55.533;
   1:  PR[GP1:91,2] = PR[GP1:90,2] + 23.484;
   1:L PR[91] 10mm/sec CNT100;
   1:  PR[GP1:91,1] = PR[GP1:90,1] + 51.838;
   1:  PR[GP1:91,2] = PR[GP1:90,2] + 27.102;
   1:L PR[91] 10mm/sec CNT100;
   1:  PR[GP1:91,1] = PR[GP1:90,1] + 48.108;
   1:  PR[GP1:91,2] = PR[GP1:90,2] + 30.478;
   1:L PR[91] 10mm/sec CNT100;
   1:  PR[GP1:91,1] = PR[GP1:90,1] + 43.820;
   1:  PR[GP1:91,2] = PR[GP1:90,2] + 33.168;
   1:L PR[91] 10mm/sec CNT100;
   1:  PR[GP1:91,1] = PR[GP1:90,1] + 38.560;
   1:  PR[GP1:91,2] = PR[GP1:90,2] + 35.466;
   1:L PR[91] 10mm/sec CNT100;
   1:  PR[GP1:91,1] = PR[GP1:90,1] + 33.957;
   1:  PR[GP1:91,2] = PR[GP1:90,2] + 37.146;
   1:L PR[91] 10mm/sec CNT100;
   1:  PR[GP1:91,1] = PR[GP1:90,1] + 29.600;
   1:  PR[GP1:91,2] = PR[GP1:90,2] + 37.764;
   1:L PR[91] 10mm/sec CNT100;
   1:  PR[GP1:91,1] = PR[GP1:90,1] + 22.891;
   1:  PR[GP1:91,2] = PR[GP1:90,2] + 38.387;
   1:L PR[91] 10mm/sec CNT100;
   1:  PR[GP1:91,1] = PR[GP1:90,1] + 18.788;
   1:  PR[GP1:91,2] = PR[GP1:90,2] + 38.115;
   1:L PR[91] 10mm/sec CNT100;
   1:  PR[GP1:91,1] = PR[GP1:90,1] + 11.426;
   1:  PR[GP1:91,2] = PR[GP1:90,2] + 36.376;
   1:L PR[91] 10mm/sec CNT100;
   1:  PR[GP1:91,1] = PR[GP1:90,1] + 7.783;
   1:  PR[GP1:91,2] = PR[GP1:90,2] + 35.329;
   1:L PR[91] 10mm/sec CNT100;
   1:  PR[GP1:91,1] = PR[GP1:90,1] + 6.768;
   1:  PR[GP1:91,2] = PR[GP1:90,2] + 34.796;
   1:L PR[91] 10mm/sec CNT100;
   1:  PR[GP1:91,1] = PR[GP1:90,1] + 4.168;
   1:  PR[GP1:91,2] = PR[GP1:90,2] + 33.393;
   1:L PR[91] 10mm/sec CNT100;
   1:  PR[GP1:91,1] = PR[GP1:90,1] + -0.263;
   1:  PR[GP1:91,2] = PR[GP1:90,2] + 29.788;
   1:L PR[91] 10mm/sec CNT100;
   1:  PR[GP1:91,1] = PR[GP1:90,1] + -4.683;
   1:  PR[GP1:91,2] = PR[GP1:90,2] + 33.382;
   1:L PR[91] 10mm/sec CNT100;
   1:  PR[GP1:91,1] = PR[GP1:90,1] + -7.299;
   1:  PR[GP1:91,2] = PR[GP1:90,2] + 34.799;
   1:L PR[91] 10mm/sec CNT100;
   1:  PR[GP1:91,1] = PR[GP1:90,1] + -8.310;
   1:  PR[GP1:91,2] = PR[GP1:90,2] + 35.330;
   1:L PR[91] 10mm/sec CNT100;
   1:  PR[GP1:91,1] = PR[GP1:90,1] + -11.949;
   1:  PR[GP1:91,2] = PR[GP1:90,2] + 36.376;
   1:L PR[91] 10mm/sec CNT100;
   1:  PR[GP1:91,1] = PR[GP1:90,1] + -19.312;
   1:  PR[GP1:91,2] = PR[GP1:90,2] + 38.115;
   1:L PR[91] 10mm/sec CNT100;
   1:  PR[GP1:91,1] = PR[GP1:90,1] + -23.414;
   1:  PR[GP1:91,2] = PR[GP1:90,2] + 38.385;
   1:L PR[91] 10mm/sec CNT100;
   1:  PR[GP1:91,1] = PR[GP1:90,1] + -28.025;
   1:  PR[GP1:91,2] = PR[GP1:90,2] + 37.747;
   1:L PR[91] 10mm/sec CNT100;
   1:  PR[GP1:91,1] = PR[GP1:90,1] + -34.521;
   1:  PR[GP1:91,2] = PR[GP1:90,2] + 37.137;
   1:L PR[91] 10mm/sec CNT100;
   1:  PR[GP1:91,1] = PR[GP1:90,1] + -39.105;
   1:  PR[GP1:91,2] = PR[GP1:90,2] + 35.458;
   1:L PR[91] 10mm/sec CNT100;
   1:  PR[GP1:91,1] = PR[GP1:90,1] + -44.364;
   1:  PR[GP1:91,2] = PR[GP1:90,2] + 33.159;
   1:L PR[91] 10mm/sec CNT100;
   1:  PR[GP1:91,1] = PR[GP1:90,1] + -48.668;
   1:  PR[GP1:91,2] = PR[GP1:90,2] + 30.444;
   1:L PR[91] 10mm/sec CNT100;
   1:  PR[GP1:91,1] = PR[GP1:90,1] + -52.575;
   1:  PR[GP1:91,2] = PR[GP1:90,2] + 26.631;
   1:L PR[91] 10mm/sec CNT100;
   1:  PR[GP1:91,1] = PR[GP1:90,1] + -56.114;
   1:  PR[GP1:91,2] = PR[GP1:90,2] + 23.427;
   1:L PR[91] 10mm/sec CNT100;
   1:  PR[GP1:91,1] = PR[GP1:90,1] + -59.146;
   1:  PR[GP1:91,2] = PR[GP1:90,2] + 18.694;
   1:L PR[91] 10mm/sec CNT100;
   1:  PR[GP1:91,1] = PR[GP1:90,1] + -61.208;
   1:  PR[GP1:91,2] = PR[GP1:90,2] + 14.970;
   1:L PR[91] 10mm/sec CNT100;
   1:  PR[GP1:91,1] = PR[GP1:90,1] + -63.130;
   1:  PR[GP1:91,2] = PR[GP1:90,2] + 9.674;
   1:L PR[91] 10mm/sec CNT100;
   1:  PR[GP1:91,1] = PR[GP1:90,1] + -63.752;
   1:  PR[GP1:91,2] = PR[GP1:90,2] + 4.122;
   1:L PR[91] 10mm/sec CNT100;
   1:  PR[GP1:91,1] = PR[GP1:90,1] + -64.412;
   1:  PR[GP1:91,2] = PR[GP1:90,2] + 0.261;
   1:L PR[91] 10mm/sec CNT100;
   1:  PR[GP1:91,1] = PR[GP1:90,1] + -63.803;
   1:  PR[GP1:91,2] = PR[GP1:90,2] + -5.205;
   1:L PR[91] 10mm/sec CNT100;
   1:  PR[GP1:91,1] = PR[GP1:90,1] + -63.139;
   1:  PR[GP1:91,2] = PR[GP1:90,2] + -9.091;
   1:L PR[91] 10mm/sec CNT100;
   1:  PR[GP1:91,1] = PR[GP1:90,1] + -61.211;
   1:  PR[GP1:91,2] = PR[GP1:90,2] + -14.403;
   1:L PR[91] 10mm/sec CNT100;
   1:  PR[GP1:91,1] = PR[GP1:90,1] + -59.158;
   1:  PR[GP1:91,2] = PR[GP1:90,2] + -18.121;
   1:L PR[91] 10mm/sec CNT100;
   1:  PR[GP1:91,1] = PR[GP1:90,1] + -56.120;
   1:  PR[GP1:91,2] = PR[GP1:90,2] + -22.863;
   1:L PR[91] 10mm/sec CNT100;
   1:  PR[GP1:91,1] = PR[GP1:90,1] + -52.419;
   1:  PR[GP1:91,2] = PR[GP1:90,2] + -26.493;
   1:L PR[91] 10mm/sec CNT100;
   1:  PR[GP1:91,1] = PR[GP1:90,1] + -48.706;
   1:  PR[GP1:91,2] = PR[GP1:90,2] + -29.862;
   1:L PR[91] 10mm/sec CNT100;
   1:  PR[GP1:91,1] = PR[GP1:90,1] + -44.393;
   1:  PR[GP1:91,2] = PR[GP1:90,2] + -32.581;
   1:L PR[91] 10mm/sec CNT100;
   1:  PR[GP1:91,1] = PR[GP1:90,1] + -39.155;
   1:  PR[GP1:91,2] = PR[GP1:90,2] + -34.886;
   1:L PR[91] 10mm/sec CNT100;
   1:  PR[GP1:91,1] = PR[GP1:90,1] + -34.560;
   1:  PR[GP1:91,2] = PR[GP1:90,2] + -36.570;
   1:L PR[91] 10mm/sec CNT100;
   1:  PR[GP1:91,1] = PR[GP1:90,1] + -30.190;
   1:  PR[GP1:91,2] = PR[GP1:90,2] + -37.192;
   1:L PR[91] 10mm/sec CNT100;
   1:  PR[GP1:91,1] = PR[GP1:90,1] + -23.503;
   1:  PR[GP1:91,2] = PR[GP1:90,2] + -37.833;
   1:L PR[91] 10mm/sec CNT100;
   1:  PR[GP1:91,1] = PR[GP1:90,1] + -19.388;
   1:  PR[GP1:91,2] = PR[GP1:90,2] + -37.562;
   1:L PR[91] 10mm/sec CNT100;
   1:  PR[GP1:91,1] = PR[GP1:90,1] + -12.146;
   1:  PR[GP1:91,2] = PR[GP1:90,2] + -35.905;
   1:L PR[91] 10mm/sec CNT100;
   1:  PR[GP1:91,1] = PR[GP1:90,1] + -8.465;
   1:  PR[GP1:91,2] = PR[GP1:90,2] + -34.847;
   1:L PR[91] 10mm/sec CNT100;
   1:  PR[GP1:91,1] = PR[GP1:90,1] + -2.275;
   1:  PR[GP1:91,2] = PR[GP1:90,2] + -31.221;
   1:L PR[91] 10mm/sec CNT100;
   1:  PR[GP1:91,1] = PR[GP1:90,1] + -1.626;
   1:  PR[GP1:91,2] = PR[GP1:90,2] + -30.868;
   1:L PR[91] 10mm/sec CNT100;
   1:  PR[GP1:91,1] = PR[GP1:90,1] + -0.265;
   1:  PR[GP1:91,2] = PR[GP1:90,2] + -29.694;
   1:L PR[91] 10mm/sec CNT100;
   1:  PR[GP1:91,1] = PR[GP1:90,1] + 0.852;
   1:  PR[GP1:91,2] = PR[GP1:90,2] + -30.939;
   1:  PR[GP1:91,3] = PR[GP1:90,3] + 66.185;
   1:L PR[91] 10mm/sec CNT100;
   1:  PR[GP1:91,1] = PR[GP1:90,1] + 1.331;
   1:  PR[GP1:91,2] = PR[GP1:90,2] + -31.199;
   1:L PR[91] 10mm/sec CNT100;
   1:  PR[GP1:91,1] = PR[GP1:90,1] + 7.680;
   1:  PR[GP1:91,2] = PR[GP1:90,2] + -34.915;
   1:L PR[91] 10mm/sec CNT100;
   1:  PR[GP1:91,1] = PR[GP1:90,1] + 11.246;
   1:  PR[GP1:91,2] = PR[GP1:90,2] + -35.939;
   1:L PR[91] 10mm/sec CNT100;
   1:  PR[GP1:91,1] = PR[GP1:90,1] + 18.687;
   1:  PR[GP1:91,2] = PR[GP1:90,2] + -37.642;
   1:L PR[91] 10mm/sec CNT100;
   1:  PR[GP1:91,1] = PR[GP1:90,1] + 22.653;
   1:  PR[GP1:91,2] = PR[GP1:90,2] + -37.905;
   1:L PR[91] 10mm/sec CNT100;
   1:  PR[GP1:91,1] = PR[GP1:90,1] + 27.110;
   1:  PR[GP1:91,2] = PR[GP1:90,2] + -37.290;
   1:L PR[91] 10mm/sec CNT100;
   1:  PR[GP1:91,1] = PR[GP1:90,1] + 33.804;
   1:  PR[GP1:91,2] = PR[GP1:90,2] + -36.639;
   1:L PR[91] 10mm/sec CNT100;
   1:  PR[GP1:91,1] = PR[GP1:90,1] + 38.266;
   1:  PR[GP1:91,2] = PR[GP1:90,2] + -35.011;
   1:L PR[91] 10mm/sec CNT100;
   1:  PR[GP1:91,1] = PR[GP1:90,1] + 43.704;
   1:  PR[GP1:91,2] = PR[GP1:90,2] + -32.619;
   1:L PR[91] 10mm/sec CNT100;
   1:  PR[GP1:91,1] = PR[GP1:90,1] + 47.871;
   1:  PR[GP1:91,2] = PR[GP1:90,2] + -30.005;
   1:L PR[91] 10mm/sec CNT100;
   1:  PR[GP1:91,1] = PR[GP1:90,1] + 51.669;
   1:  PR[GP1:91,2] = PR[GP1:90,2] + -26.303;
   1:L PR[91] 10mm/sec CNT100;
   1:  PR[GP1:91,1] = PR[GP1:90,1] + 55.365;
   1:  PR[GP1:91,2] = PR[GP1:90,2] + -22.942;
   1:L PR[91] 10mm/sec CNT100;
   1:  PR[GP1:91,1] = PR[GP1:90,1] + 58.355;
   1:  PR[GP1:91,2] = PR[GP1:90,2] + -18.304;
   1:L PR[91] 10mm/sec CNT100;
   1:  PR[GP1:91,1] = PR[GP1:90,1] + 60.516;
   1:  PR[GP1:91,2] = PR[GP1:90,2] + -14.398;
   1:L PR[91] 10mm/sec CNT100;
   1:  PR[GP1:91,1] = PR[GP1:90,1] + 62.384;
   1:  PR[GP1:91,2] = PR[GP1:90,2] + -9.317;
   1:L PR[91] 10mm/sec CNT100;
   1:  PR[GP1:91,1] = PR[GP1:90,1] + 63.014;
   1:  PR[GP1:91,2] = PR[GP1:90,2] + -3.780;
   1:L PR[91] 10mm/sec CNT100;
   1:  PR[GP1:91,1] = PR[GP1:90,1] + 63.709;
   1:  PR[GP1:91,2] = PR[GP1:90,2] + 0.296;
   1:L PR[91] 10mm/sec CNT100;
   1:  PR[GP1:91,1] = PR[GP1:90,1] + 63.092;
   1:  PR[GP1:91,2] = PR[GP1:90,2] + 5.751;
   1:L PR[91] 10mm/sec CNT100;
   1:  PR[GP1:91,1] = PR[GP1:90,1] + 62.387;
   1:  PR[GP1:91,2] = PR[GP1:90,2] + 9.868;
   1:L PR[91] 10mm/sec CNT100;
   1:  PR[GP1:91,1] = PR[GP1:90,1] + 60.513;
   1:  PR[GP1:91,2] = PR[GP1:90,2] + 14.965;
   1:L PR[91] 10mm/sec CNT100;
   1:  PR[GP1:91,1] = PR[GP1:90,1] + 58.342;
   1:  PR[GP1:91,2] = PR[GP1:90,2] + 18.878;
   1:L PR[91] 10mm/sec CNT100;
   1:  PR[GP1:91,1] = PR[GP1:90,1] + 55.346;
   1:  PR[GP1:91,2] = PR[GP1:90,2] + 23.526;
   1:L PR[91] 10mm/sec CNT100;
   1:  PR[GP1:91,1] = PR[GP1:90,1] + 51.741;
   1:  PR[GP1:91,2] = PR[GP1:90,2] + 27.056;
   1:L PR[91] 10mm/sec CNT100;
   1:  PR[GP1:91,1] = PR[GP1:90,1] + 47.851;
   1:  PR[GP1:91,2] = PR[GP1:90,2] + 30.576;
   1:L PR[91] 10mm/sec CNT100;
   1:  PR[GP1:91,1] = PR[GP1:90,1] + 43.674;
   1:  PR[GP1:91,2] = PR[GP1:90,2] + 33.197;
   1:L PR[91] 10mm/sec CNT100;
   1:  PR[GP1:91,1] = PR[GP1:90,1] + 38.215;
   1:  PR[GP1:91,2] = PR[GP1:90,2] + 35.582;
   1:L PR[91] 10mm/sec CNT100;
   1:  PR[GP1:91,1] = PR[GP1:90,1] + 33.738;
   1:  PR[GP1:91,2] = PR[GP1:90,2] + 37.216;
   1:L PR[91] 10mm/sec CNT100;
   1:  PR[GP1:91,1] = PR[GP1:90,1] + 29.500;
   1:  PR[GP1:91,2] = PR[GP1:90,2] + 37.817;
   1:L PR[91] 10mm/sec CNT100;
   1:  PR[GP1:91,1] = PR[GP1:90,1] + 22.588;
   1:  PR[GP1:91,2] = PR[GP1:90,2] + 38.459;
   1:L PR[91] 10mm/sec CNT100;
   1:  PR[GP1:91,1] = PR[GP1:90,1] + 18.609;
   1:  PR[GP1:91,2] = PR[GP1:90,2] + 38.195;
   1:L PR[91] 10mm/sec CNT100;
   1:  PR[GP1:91,1] = PR[GP1:90,1] + 11.046;
   1:  PR[GP1:91,2] = PR[GP1:90,2] + 36.409;
   1:L PR[91] 10mm/sec CNT100;
   1:  PR[GP1:91,1] = PR[GP1:90,1] + 7.525;
   1:  PR[GP1:91,2] = PR[GP1:90,2] + 35.396;
   1:L PR[91] 10mm/sec CNT100;
   1:  PR[GP1:91,1] = PR[GP1:90,1] + 6.484;
   1:  PR[GP1:91,2] = PR[GP1:90,2] + 34.851;
   1:L PR[91] 10mm/sec CNT100;
   1:  PR[GP1:91,1] = PR[GP1:90,1] + 3.995;
   1:  PR[GP1:91,2] = PR[GP1:90,2] + 33.507;
   1:L PR[91] 10mm/sec CNT100;
   1:  PR[GP1:91,1] = PR[GP1:90,1] + -0.263;
   1:  PR[GP1:91,2] = PR[GP1:90,2] + 30.043;
   1:L PR[91] 10mm/sec CNT100;
   1:  PR[GP1:91,1] = PR[GP1:90,1] + -4.511;
   1:  PR[GP1:91,2] = PR[GP1:90,2] + 33.497;
   1:L PR[91] 10mm/sec CNT100;
   1:  PR[GP1:91,1] = PR[GP1:90,1] + -7.014;
   1:  PR[GP1:91,2] = PR[GP1:90,2] + 34.852;
   1:L PR[91] 10mm/sec CNT100;
   1:  PR[GP1:91,1] = PR[GP1:90,1] + -8.052;
   1:  PR[GP1:91,2] = PR[GP1:90,2] + 35.398;
   1:L PR[91] 10mm/sec CNT100;
   1:  PR[GP1:91,1] = PR[GP1:90,1] + -11.568;
   1:  PR[GP1:91,2] = PR[GP1:90,2] + 36.409;
   1:L PR[91] 10mm/sec CNT100;
   1:  PR[GP1:91,1] = PR[GP1:90,1] + -19.133;
   1:  PR[GP1:91,2] = PR[GP1:90,2] + 38.195;
   1:L PR[91] 10mm/sec CNT100;
   1:  PR[GP1:91,1] = PR[GP1:90,1] + -23.112;
   1:  PR[GP1:91,2] = PR[GP1:90,2] + 38.457;
   1:L PR[91] 10mm/sec CNT100;
   1:  PR[GP1:91,1] = PR[GP1:90,1] + -27.586;
   1:  PR[GP1:91,2] = PR[GP1:90,2] + 37.838;
   1:L PR[91] 10mm/sec CNT100;
   1:  PR[GP1:91,1] = PR[GP1:90,1] + -34.301;
   1:  PR[GP1:91,2] = PR[GP1:90,2] + 37.207;
   1:L PR[91] 10mm/sec CNT100;
   1:  PR[GP1:91,1] = PR[GP1:90,1] + -38.759;
   1:  PR[GP1:91,2] = PR[GP1:90,2] + 35.574;
   1:L PR[91] 10mm/sec CNT100;
   1:  PR[GP1:91,1] = PR[GP1:90,1] + -44.217;
   1:  PR[GP1:91,2] = PR[GP1:90,2] + 33.188;
   1:L PR[91] 10mm/sec CNT100;
   1:  PR[GP1:91,1] = PR[GP1:90,1] + -48.410;
   1:  PR[GP1:91,2] = PR[GP1:90,2] + 30.544;
   1:L PR[91] 10mm/sec CNT100;
   1:  PR[GP1:91,1] = PR[GP1:90,1] + -52.217;
   1:  PR[GP1:91,2] = PR[GP1:90,2] + 26.828;
   1:L PR[91] 10mm/sec CNT100;
   1:  PR[GP1:91,1] = PR[GP1:90,1] + -55.925;
   1:  PR[GP1:91,2] = PR[GP1:90,2] + 23.470;
   1:L PR[91] 10mm/sec CNT100;
   1:  PR[GP1:91,1] = PR[GP1:90,1] + -58.883;
   1:  PR[GP1:91,2] = PR[GP1:90,2] + 18.853;
   1:L PR[91] 10mm/sec CNT100;
   1:  PR[GP1:91,1] = PR[GP1:90,1] + -61.053;
   1:  PR[GP1:91,2] = PR[GP1:90,2] + 14.934;
   1:L PR[91] 10mm/sec CNT100;
   1:  PR[GP1:91,1] = PR[GP1:90,1] + -62.930;
   1:  PR[GP1:91,2] = PR[GP1:90,2] + 9.763;
   1:L PR[91] 10mm/sec CNT100;
   1:  PR[GP1:91,1] = PR[GP1:90,1] + -63.537;
   1:  PR[GP1:91,2] = PR[GP1:90,2] + 4.342;
   1:L PR[91] 10mm/sec CNT100;
   1:  PR[GP1:91,1] = PR[GP1:90,1] + -64.235;
   1:  PR[GP1:91,2] = PR[GP1:90,2] + 0.261;
   1:L PR[91] 10mm/sec CNT100;
   1:  PR[GP1:91,1] = PR[GP1:90,1] + -63.640;
   1:  PR[GP1:91,2] = PR[GP1:90,2] + -5.078;
   1:L PR[91] 10mm/sec CNT100;
   1:  PR[GP1:91,1] = PR[GP1:90,1] + -62.939;
   1:  PR[GP1:91,2] = PR[GP1:90,2] + -9.180;
   1:L PR[91] 10mm/sec CNT100;
   1:  PR[GP1:91,1] = PR[GP1:90,1] + -61.056;
   1:  PR[GP1:91,2] = PR[GP1:90,2] + -14.367;
   1:L PR[91] 10mm/sec CNT100;
   1:  PR[GP1:91,1] = PR[GP1:90,1] + -58.896;
   1:  PR[GP1:91,2] = PR[GP1:90,2] + -18.279;
   1:L PR[91] 10mm/sec CNT100;
   1:  PR[GP1:91,1] = PR[GP1:90,1] + -55.931;
   1:  PR[GP1:91,2] = PR[GP1:90,2] + -22.906;
   1:L PR[91] 10mm/sec CNT100;
   1:  PR[GP1:91,1] = PR[GP1:90,1] + -52.321;
   1:  PR[GP1:91,2] = PR[GP1:90,2] + -26.448;
   1:L PR[91] 10mm/sec CNT100;
   1:  PR[GP1:91,1] = PR[GP1:90,1] + -48.450;
   1:  PR[GP1:91,2] = PR[GP1:90,2] + -29.960;
   1:L PR[91] 10mm/sec CNT100;
   1:  PR[GP1:91,1] = PR[GP1:90,1] + -44.248;
   1:  PR[GP1:91,2] = PR[GP1:90,2] + -32.610;
   1:L PR[91] 10mm/sec CNT100;
   1:  PR[GP1:91,1] = PR[GP1:90,1] + -38.811;
   1:  PR[GP1:91,2] = PR[GP1:90,2] + -35.002;
   1:L PR[91] 10mm/sec CNT100;
   1:  PR[GP1:91,1] = PR[GP1:90,1] + -34.342;
   1:  PR[GP1:91,2] = PR[GP1:90,2] + -36.640;
   1:L PR[91] 10mm/sec CNT100;
   1:  PR[GP1:91,1] = PR[GP1:90,1] + -30.092;
   1:  PR[GP1:91,2] = PR[GP1:90,2] + -37.244;
   1:L PR[91] 10mm/sec CNT100;
   1:  PR[GP1:91,1] = PR[GP1:90,1] + -23.203;
   1:  PR[GP1:91,2] = PR[GP1:90,2] + -37.905;
   1:L PR[91] 10mm/sec CNT100;
   1:  PR[GP1:91,1] = PR[GP1:90,1] + -19.212;
   1:  PR[GP1:91,2] = PR[GP1:90,2] + -37.642;
   1:L PR[91] 10mm/sec CNT100;
   1:  PR[GP1:91,1] = PR[GP1:90,1] + -11.771;
   1:  PR[GP1:91,2] = PR[GP1:90,2] + -35.939;
   1:L PR[91] 10mm/sec CNT100;
   1:  PR[GP1:91,1] = PR[GP1:90,1] + -8.210;
   1:  PR[GP1:91,2] = PR[GP1:90,2] + -34.917;
   1:L PR[91] 10mm/sec CNT100;
   1:  PR[GP1:91,1] = PR[GP1:90,1] + -1.865;
   1:  PR[GP1:91,2] = PR[GP1:90,2] + -31.199;
   1:L PR[91] 10mm/sec CNT100;
   1:  PR[GP1:91,1] = PR[GP1:90,1] + -1.383;
   1:  PR[GP1:91,2] = PR[GP1:90,2] + -30.937;
   1:L PR[91] 10mm/sec CNT100;
   1:  PR[GP1:91,1] = PR[GP1:90,1] + -0.266;
   1:  PR[GP1:91,2] = PR[GP1:90,2] + -29.973;
   1:L PR[91] 10mm/sec CNT100;
   1:  PR[GP1:91,1] = PR[GP1:90,1] + 0.608;
   1:  PR[GP1:91,2] = PR[GP1:90,2] + -31.007;
   1:  PR[GP1:91,3] = PR[GP1:90,3] + 66.795;
   1:L PR[91] 10mm/sec CNT100;
   1:  PR[GP1:91,1] = PR[GP1:90,1] + 0.920;
   1:  PR[GP1:91,2] = PR[GP1:90,2] + -31.177;
   1:L PR[91] 10mm/sec CNT100;
   1:  PR[GP1:91,1] = PR[GP1:90,1] + 7.425;
   1:  PR[GP1:91,2] = PR[GP1:90,2] + -34.985;
   1:L PR[91] 10mm/sec CNT100;
   1:  PR[GP1:91,1] = PR[GP1:90,1] + 10.870;
   1:  PR[GP1:91,2] = PR[GP1:90,2] + -35.974;
   1:L PR[91] 10mm/sec CNT100;
   1:  PR[GP1:91,1] = PR[GP1:90,1] + 18.510;
   1:  PR[GP1:91,2] = PR[GP1:90,2] + -37.722;
   1:L PR[91] 10mm/sec CNT100;
   1:  PR[GP1:91,1] = PR[GP1:90,1] + 22.353;
   1:  PR[GP1:91,2] = PR[GP1:90,2] + -37.977;
   1:L PR[91] 10mm/sec CNT100;
   1:  PR[GP1:91,1] = PR[GP1:90,1] + 26.674;
   1:  PR[GP1:91,2] = PR[GP1:90,2] + -37.381;
   1:L PR[91] 10mm/sec CNT100;
   1:  PR[GP1:91,1] = PR[GP1:90,1] + 33.587;
   1:  PR[GP1:91,2] = PR[GP1:90,2] + -36.709;
   1:L PR[91] 10mm/sec CNT100;
   1:  PR[GP1:91,1] = PR[GP1:90,1] + 37.922;
   1:  PR[GP1:91,2] = PR[GP1:90,2] + -35.127;
   1:L PR[91] 10mm/sec CNT100;
   1:  PR[GP1:91,1] = PR[GP1:90,1] + 43.559;
   1:  PR[GP1:91,2] = PR[GP1:90,2] + -32.648;
   1:L PR[91] 10mm/sec CNT100;
   1:  PR[GP1:91,1] = PR[GP1:90,1] + 47.616;
   1:  PR[GP1:91,2] = PR[GP1:90,2] + -30.102;
   1:L PR[91] 10mm/sec CNT100;
   1:  PR[GP1:91,1] = PR[GP1:90,1] + 51.314;
   1:  PR[GP1:91,2] = PR[GP1:90,2] + -26.498;
   1:L PR[91] 10mm/sec CNT100;
   1:  PR[GP1:91,1] = PR[GP1:90,1] + 55.178;
   1:  PR[GP1:91,2] = PR[GP1:90,2] + -22.983;
   1:L PR[91] 10mm/sec CNT100;
   1:  PR[GP1:91,1] = PR[GP1:90,1] + 58.093;
   1:  PR[GP1:91,2] = PR[GP1:90,2] + -18.462;
   1:L PR[91] 10mm/sec CNT100;
   1:  PR[GP1:91,1] = PR[GP1:90,1] + 60.362;
   1:  PR[GP1:91,2] = PR[GP1:90,2] + -14.361;
   1:L PR[91] 10mm/sec CNT100;
   1:  PR[GP1:91,1] = PR[GP1:90,1] + 62.185;
   1:  PR[GP1:91,2] = PR[GP1:90,2] + -9.404;
   1:L PR[91] 10mm/sec CNT100;
   1:  PR[GP1:91,1] = PR[GP1:90,1] + 62.799;
   1:  PR[GP1:91,2] = PR[GP1:90,2] + -3.999;
   1:L PR[91] 10mm/sec CNT100;
   1:  PR[GP1:91,1] = PR[GP1:90,1] + 63.532;
   1:  PR[GP1:91,2] = PR[GP1:90,2] + 0.296;
   1:L PR[91] 10mm/sec CNT100;
   1:  PR[GP1:91,1] = PR[GP1:90,1] + 62.930;
   1:  PR[GP1:91,2] = PR[GP1:90,2] + 5.621;
   1:L PR[91] 10mm/sec CNT100;
   1:  PR[GP1:91,1] = PR[GP1:90,1] + 62.187;
   1:  PR[GP1:91,2] = PR[GP1:90,2] + 9.955;
   1:L PR[91] 10mm/sec CNT100;
   1:  PR[GP1:91,1] = PR[GP1:90,1] + 60.358;
   1:  PR[GP1:91,2] = PR[GP1:90,2] + 14.928;
   1:L PR[91] 10mm/sec CNT100;
   1:  PR[GP1:91,1] = PR[GP1:90,1] + 58.080;
   1:  PR[GP1:91,2] = PR[GP1:90,2] + 19.036;
   1:L PR[91] 10mm/sec CNT100;
   1:  PR[GP1:91,1] = PR[GP1:90,1] + 55.158;
   1:  PR[GP1:91,2] = PR[GP1:90,2] + 23.568;
   1:L PR[91] 10mm/sec CNT100;
   1:  PR[GP1:91,1] = PR[GP1:90,1] + 51.643;
   1:  PR[GP1:91,2] = PR[GP1:90,2] + 27.010;
   1:L PR[91] 10mm/sec CNT100;
   1:  PR[GP1:91,1] = PR[GP1:90,1] + 47.594;
   1:  PR[GP1:91,2] = PR[GP1:90,2] + 30.674;
   1:L PR[91] 10mm/sec CNT100;
   1:  PR[GP1:91,1] = PR[GP1:90,1] + 43.527;
   1:  PR[GP1:91,2] = PR[GP1:90,2] + 33.226;
   1:L PR[91] 10mm/sec CNT100;
   1:  PR[GP1:91,1] = PR[GP1:90,1] + 37.869;
   1:  PR[GP1:91,2] = PR[GP1:90,2] + 35.699;
   1:L PR[91] 10mm/sec CNT100;
   1:  PR[GP1:91,1] = PR[GP1:90,1] + 33.518;
   1:  PR[GP1:91,2] = PR[GP1:90,2] + 37.286;
   1:L PR[91] 10mm/sec CNT100;
   1:  PR[GP1:91,1] = PR[GP1:90,1] + 29.401;
   1:  PR[GP1:91,2] = PR[GP1:90,2] + 37.870;
   1:L PR[91] 10mm/sec CNT100;
   1:  PR[GP1:91,1] = PR[GP1:90,1] + 22.286;
   1:  PR[GP1:91,2] = PR[GP1:90,2] + 38.531;
   1:L PR[91] 10mm/sec CNT100;
   1:  PR[GP1:91,1] = PR[GP1:90,1] + 18.430;
   1:  PR[GP1:91,2] = PR[GP1:90,2] + 38.275;
   1:L PR[91] 10mm/sec CNT100;
   1:  PR[GP1:91,1] = PR[GP1:90,1] + 10.665;
   1:  PR[GP1:91,2] = PR[GP1:90,2] + 36.441;
   1:L PR[91] 10mm/sec CNT100;
   1:  PR[GP1:91,1] = PR[GP1:90,1] + 7.267;
   1:  PR[GP1:91,2] = PR[GP1:90,2] + 35.464;
   1:L PR[91] 10mm/sec CNT100;
   1:  PR[GP1:91,1] = PR[GP1:90,1] + 6.199;
   1:  PR[GP1:91,2] = PR[GP1:90,2] + 34.904;
   1:L PR[91] 10mm/sec CNT100;
   1:  PR[GP1:91,1] = PR[GP1:90,1] + 3.823;
   1:  PR[GP1:91,2] = PR[GP1:90,2] + 33.621;
   1:L PR[91] 10mm/sec CNT100;
   1:  PR[GP1:91,1] = PR[GP1:90,1] + -0.263;
   1:  PR[GP1:91,2] = PR[GP1:90,2] + 30.298;
   1:L PR[91] 10mm/sec CNT100;
   1:  PR[GP1:91,1] = PR[GP1:90,1] + -4.339;
   1:  PR[GP1:91,2] = PR[GP1:90,2] + 33.611;
   1:L PR[91] 10mm/sec CNT100;
   1:  PR[GP1:91,1] = PR[GP1:90,1] + -6.728;
   1:  PR[GP1:91,2] = PR[GP1:90,2] + 34.905;
   1:L PR[91] 10mm/sec CNT100;
   1:  PR[GP1:91,1] = PR[GP1:90,1] + -7.794;
   1:  PR[GP1:91,2] = PR[GP1:90,2] + 35.466;
   1:L PR[91] 10mm/sec CNT100;
   1:  PR[GP1:91,1] = PR[GP1:90,1] + -11.187;
   1:  PR[GP1:91,2] = PR[GP1:90,2] + 36.441;
   1:L PR[91] 10mm/sec CNT100;
   1:  PR[GP1:91,1] = PR[GP1:90,1] + -18.954;
   1:  PR[GP1:91,2] = PR[GP1:90,2] + 38.275;
   1:L PR[91] 10mm/sec CNT100;
   1:  PR[GP1:91,1] = PR[GP1:90,1] + -22.809;
   1:  PR[GP1:91,2] = PR[GP1:90,2] + 38.529;
   1:L PR[91] 10mm/sec CNT100;
   1:  PR[GP1:91,1] = PR[GP1:90,1] + -27.147;
   1:  PR[GP1:91,2] = PR[GP1:90,2] + 37.929;
   1:L PR[91] 10mm/sec CNT100;
   1:  PR[GP1:91,1] = PR[GP1:90,1] + -34.081;
   1:  PR[GP1:91,2] = PR[GP1:90,2] + 37.277;
   1:L PR[91] 10mm/sec CNT100;
   1:  PR[GP1:91,1] = PR[GP1:90,1] + -38.412;
   1:  PR[GP1:91,2] = PR[GP1:90,2] + 35.691;
   1:L PR[91] 10mm/sec CNT100;
   1:  PR[GP1:91,1] = PR[GP1:90,1] + -44.070;
   1:  PR[GP1:91,2] = PR[GP1:90,2] + 33.217;
   1:L PR[91] 10mm/sec CNT100;
   1:  PR[GP1:91,1] = PR[GP1:90,1] + -48.152;
   1:  PR[GP1:91,2] = PR[GP1:90,2] + 30.643;
   1:L PR[91] 10mm/sec CNT100;
   1:  PR[GP1:91,1] = PR[GP1:90,1] + -51.859;
   1:  PR[GP1:91,2] = PR[GP1:90,2] + 27.024;
   1:L PR[91] 10mm/sec CNT100;
   1:  PR[GP1:91,1] = PR[GP1:90,1] + -55.736;
   1:  PR[GP1:91,2] = PR[GP1:90,2] + 23.514;
   1:L PR[91] 10mm/sec CNT100;
   1:  PR[GP1:91,1] = PR[GP1:90,1] + -58.621;
   1:  PR[GP1:91,2] = PR[GP1:90,2] + 19.012;
   1:L PR[91] 10mm/sec CNT100;
   1:  PR[GP1:91,1] = PR[GP1:90,1] + -60.898;
   1:  PR[GP1:91,2] = PR[GP1:90,2] + 14.898;
   1:L PR[91] 10mm/sec CNT100;
   1:  PR[GP1:91,1] = PR[GP1:90,1] + -62.729;
   1:  PR[GP1:91,2] = PR[GP1:90,2] + 9.853;
   1:L PR[91] 10mm/sec CNT100;
   1:  PR[GP1:91,1] = PR[GP1:90,1] + -63.322;
   1:  PR[GP1:91,2] = PR[GP1:90,2] + 4.562;
   1:L PR[91] 10mm/sec CNT100;
   1:  PR[GP1:91,1] = PR[GP1:90,1] + -64.058;
   1:  PR[GP1:91,2] = PR[GP1:90,2] + 0.261;
   1:L PR[91] 10mm/sec CNT100;
   1:  PR[GP1:91,1] = PR[GP1:90,1] + -63.477;
   1:  PR[GP1:91,2] = PR[GP1:90,2] + -4.950;
   1:L PR[91] 10mm/sec CNT100;
   1:  PR[GP1:91,1] = PR[GP1:90,1] + -62.739;
   1:  PR[GP1:91,2] = PR[GP1:90,2] + -9.270;
   1:L PR[91] 10mm/sec CNT100;
   1:  PR[GP1:91,1] = PR[GP1:90,1] + -60.902;
   1:  PR[GP1:91,2] = PR[GP1:90,2] + -14.331;
   1:L PR[91] 10mm/sec CNT100;
   1:  PR[GP1:91,1] = PR[GP1:90,1] + -58.634;
   1:  PR[GP1:91,2] = PR[GP1:90,2] + -18.438;
   1:L PR[91] 10mm/sec CNT100;
   1:  PR[GP1:91,1] = PR[GP1:90,1] + -55.743;
   1:  PR[GP1:91,2] = PR[GP1:90,2] + -22.949;
   1:L PR[91] 10mm/sec CNT100;
   1:  PR[GP1:91,1] = PR[GP1:90,1] + -52.223;
   1:  PR[GP1:91,2] = PR[GP1:90,2] + -26.402;
   1:L PR[91] 10mm/sec CNT100;
   1:  PR[GP1:91,1] = PR[GP1:90,1] + -48.193;
   1:  PR[GP1:91,2] = PR[GP1:90,2] + -30.059;
   1:L PR[91] 10mm/sec CNT100;
   1:  PR[GP1:91,1] = PR[GP1:90,1] + -44.102;
   1:  PR[GP1:91,2] = PR[GP1:90,2] + -32.638;
   1:L PR[91] 10mm/sec CNT100;
   1:  PR[GP1:91,1] = PR[GP1:90,1] + -38.466;
   1:  PR[GP1:91,2] = PR[GP1:90,2] + -35.119;
   1:L PR[91] 10mm/sec CNT100;
   1:  PR[GP1:91,1] = PR[GP1:90,1] + -34.124;
   1:  PR[GP1:91,2] = PR[GP1:90,2] + -36.709;
   1:L PR[91] 10mm/sec CNT100;
   1:  PR[GP1:91,1] = PR[GP1:90,1] + -29.994;
   1:  PR[GP1:91,2] = PR[GP1:90,2] + -37.297;
   1:L PR[91] 10mm/sec CNT100;
   1:  PR[GP1:91,1] = PR[GP1:90,1] + -22.903;
   1:  PR[GP1:91,2] = PR[GP1:90,2] + -37.977;
   1:L PR[91] 10mm/sec CNT100;
   1:  PR[GP1:91,1] = PR[GP1:90,1] + -19.035;
   1:  PR[GP1:91,2] = PR[GP1:90,2] + -37.722;
   1:L PR[91] 10mm/sec CNT100;
   1:  PR[GP1:91,1] = PR[GP1:90,1] + -11.395;
   1:  PR[GP1:91,2] = PR[GP1:90,2] + -35.974;
   1:L PR[91] 10mm/sec CNT100;
   1:  PR[GP1:91,1] = PR[GP1:90,1] + -7.955;
   1:  PR[GP1:91,2] = PR[GP1:90,2] + -34.986;
   1:L PR[91] 10mm/sec CNT100;
   1:  PR[GP1:91,1] = PR[GP1:90,1] + -1.454;
   1:  PR[GP1:91,2] = PR[GP1:90,2] + -31.178;
   1:L PR[91] 10mm/sec CNT100;
   1:  PR[GP1:91,1] = PR[GP1:90,1] + -1.139;
